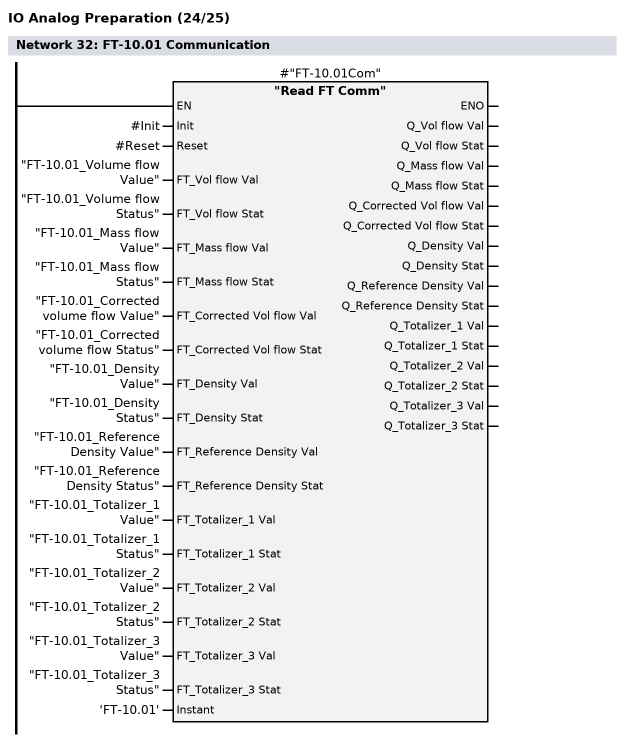
   RUNG wire#powerrail
      #"FT-10.01Com"(Init := #Init, Reset := #Reset, "FT_Vol flow Val" := "FT-10.01_Volume flow Value", "FT_Vol flow Stat" := "FT-10.01_Volume flow Status", "FT_Mass flow Val" := "FT-10.01_Mass flow Value", "FT_Mass flow Stat" := "FT-10.01_Mass flow Status", "FT_Corrected Vol flow Val" := "FT-10.01_Corrected volume flow Value", "FT_Corrected Vol flow Stat" := "FT-10.01_Corrected volume flow Status", "FT_Density Val" := "FT-10.01_Density Value", "FT_Density Stat" := "FT-10.01_Density Status", "FT_Reference Density Val" := "FT-10.01_Reference Density Value", "FT_Reference Density Stat" := "FT-10.01_Reference Density Status", "FT_Totalizer_1 Val" := "FT-10.01_Totalizer_1 Value", "FT_Totalizer_1 Stat" := "FT-10.01_Totalizer_1 Status", "FT_Totalizer_2 Val" := "FT-10.01_Totalizer_2 Value", "FT_Totalizer_2 Stat" := "FT-10.01_Totalizer_2 Status", "FT_Totalizer_3 Val" := "FT-10.01_Totalizer_3 Value", "FT_Totalizer_3 Stat" := "FT-10.01_Totalizer_3 Status", Instant := 'FT-10.01', "Q_Vol flow Val" =>, "Q_Vol flow Stat" =>, "Q_Mass flow Val" =>, "Q_Mass flow Stat" =>, "Q_Corrected Vol flow Val" =>, "Q_Corrected Vol flow Stat" =>, "Q_Density Val" =>, "Q_Density Stat" =>, "Q_Reference Density Val" =>, "Q_Reference Density Stat" =>, "Q_Totalizer_1 Val" =>, "Q_Totalizer_1 Stat" =>, "Q_Totalizer_2 Val" =>, "Q_Totalizer_2 Stat" =>, "Q_Totalizer_3 Val" =>, "Q_Totalizer_3 Stat" =>)
   END_RUNG
   // the same network as SCL:
   #"FT-10.01Com"(Init := #Init,   // "Read FT Comm"
                  Reset := #Reset,
                  "FT_Vol flow Val" := "FT-10.01_Volume flow Value",
                  "FT_Vol flow Stat" := "FT-10.01_Volume flow Status",
                  "FT_Mass flow Val" := "FT-10.01_Mass flow Value",
                  "FT_Mass flow Stat" := "FT-10.01_Mass flow Status",
                  "FT_Corrected Vol flow Val" := "FT-10.01_Corrected volume flow Value",
                  "FT_Corrected Vol flow Stat" := "FT-10.01_Corrected volume flow Status",
                  "FT_Density Val" := "FT-10.01_Density Value",
                  "FT_Density Stat" := "FT-10.01_Density Status",
                  "FT_Reference Density Val" := "FT-10.01_Reference Density Value",
                  "FT_Reference Density Stat" := "FT-10.01_Reference Density Status",
                  "FT_Totalizer_1 Val" := "FT-10.01_Totalizer_1 Value",
                  "FT_Totalizer_1 Stat" := "FT-10.01_Totalizer_1 Status",
                  "FT_Totalizer_2 Val" := "FT-10.01_Totalizer_2 Value",
                  "FT_Totalizer_2 Stat" := "FT-10.01_Totalizer_2 Status",
                  "FT_Totalizer_3 Val" := "FT-10.01_Totalizer_3 Value",
                  "FT_Totalizer_3 Stat" := "FT-10.01_Totalizer_3 Status",
                  Instant := 'FT-10.01');
END_REGION

REGION Network 33: FT-10.01 Flowrate
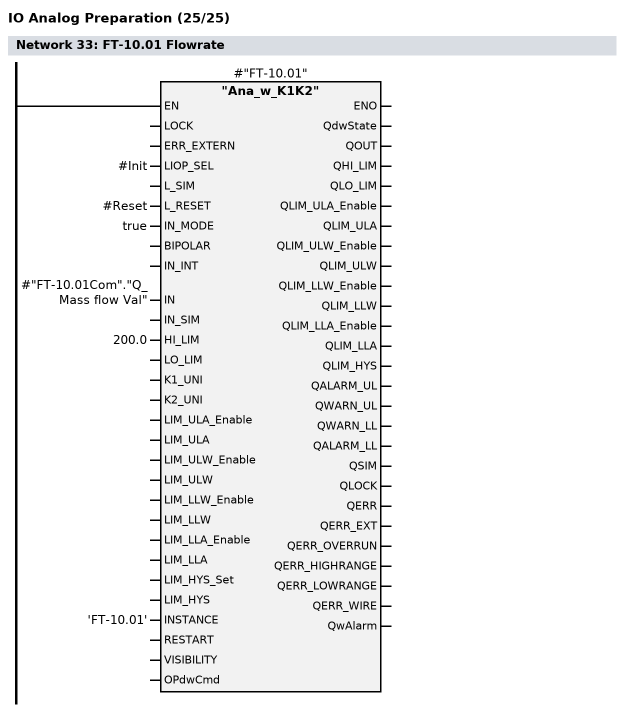
   RUNG wire#powerrail
      #"FT-10.01"(LOCK :=, ERR_EXTERN :=, LIOP_SEL := #Init, L_SIM :=, L_RESET := #Reset, IN_MODE := true, BIPOLAR :=, IN_INT :=, IN := #"FT-10.01Com"."Q_Mass flow Val", IN_SIM :=, HI_LIM := 200.0, LO_LIM :=, K1_UNI :=, K2_UNI :=, LIM_ULA_Enable :=, LIM_ULA :=, LIM_ULW_Enable :=, LIM_ULW :=, LIM_LLW_Enable :=, LIM_LLW :=, LIM_LLA_Enable :=, LIM_LLA :=, LIM_HYS_Set :=, LIM_HYS :=, INSTANCE := 'FT-10.01', RESTART :=, VISIBILITY :=, OPdwCmd :=, QdwState =>, QOUT =>, QHI_LIM =>, QLO_LIM =>, QLIM_ULA_Enable =>, QLIM_ULA =>, QLIM_ULW_Enable =>, QLIM_ULW =>, QLIM_LLW_Enable =>, QLIM_LLW =>, QLIM_LLA_Enable =>, QLIM_LLA =>, QLIM_HYS =>, QALARM_UL =>, QWARN_UL =>, QWARN_LL =>, QALARM_LL =>, QSIM =>, QLOCK =>, QERR =>, QERR_EXT =>, QERR_OVERRUN =>, QERR_HIGHRANGE =>, QERR_LOWRANGE =>, QERR_WIRE =>, QwAlarm =>)
   END_RUNG
   // the same network as SCL:
   #"FT-10.01"(LIOP_SEL := #Init,   // "Ana_w_K1K2"
               L_RESET := #Reset,
               IN_MODE := true,
               IN := #"FT-10.01Com"."Q_Mass flow Val",
               HI_LIM := 200.0,
               INSTANCE := 'FT-10.01');
END_REGION
END_FUNCTION_BLOCK

FUNCTION_BLOCK "Read FT Comm"   // FB642, LAD
{ S7_Optimized_Access := 'FALSE' }
VERSION : 0.1
// stored: AutoNumber false, IsIECCheckEnabled false, SetENOAutomatically false, UDAEnableTagReadback false
   VAR_INPUT
      Init : Bool;
      Reset : Bool;
      "FT_Vol flow Val" : Real;   // FT_Volume flow Value
      "FT_Vol flow Stat" : Byte;   // FT_Volume flow Status
      "FT_Mass flow Val" : Real;   // FT_Mass flow Value
      "FT_Mass flow Stat" : Byte;   // FT_Mass flow Status
      "FT_Corrected Vol flow Val" : Real;   // FT_Corrected volume flow Value
      "FT_Corrected Vol flow Stat" : Byte;   // FT_Corrected volume flow Status
      "FT_Density Val" : Real;   // FT_Velocity Value
      "FT_Density Stat" : Byte;   // FT_Velocity Status
      "FT_Reference Density Val" : Real;
      "FT_Reference Density Stat" : Byte;
      "FT_Totalizer_1 Val" : Real;   // FT_Totalizer_1 Value
      "FT_Totalizer_1 Stat" : Byte;   // FT_Totalizer_1 Status
      "FT_Totalizer_2 Val" : Real;   // FT_Totalizer_2 Value
      "FT_Totalizer_2 Stat" : Byte;   // FT_Totalizer_2 Status
      "FT_Totalizer_3 Val" : Real;   // FT_Totalizer_3 Value
      "FT_Totalizer_3 Stat" : Byte;   // FT_Totalizer_3 Status
      Instant { ExternalAccessible := 'False'; ExternalVisible := 'False'; ExternalWritable := 'False'} : String;
   END_VAR
   VAR_OUTPUT
      "Q_Vol flow Val" : Real;   // FT_Volume flow Value
      "Q_Vol flow Stat" : Word;   // FT_Volume flow Status
      "Q_Mass flow Val" : Real;   // FT_Mass flow Value
      "Q_Mass flow Stat" : Word;   // FT_Mass flow Status
      "Q_Corrected Vol flow Val" : Real;   // FT_Corrected volume flow Value
      "Q_Corrected Vol flow Stat" : Word;   // FT_Corrected volume flow Status
      "Q_Density Val" : Real;   // FT_Velocity Value
      "Q_Density Stat" : Word;   // FT_Velocity Status
      "Q_Reference Density Val" : Real;
      "Q_Reference Density Stat" : Word;
      "Q_Totalizer_1 Val" : Real;   // FT_Totalizer_1 Value
      "Q_Totalizer_1 Stat" : Word;   // FT_Totalizer_1 Status
      "Q_Totalizer_2 Val" : Real;   // FT_Totalizer_2 Value
      "Q_Totalizer_2 Stat" : Word;   // FT_Totalizer_2 Status
      "Q_Totalizer_3 Val" : Real;   // FT_Totalizer_3 Value
      "Q_Totalizer_3 Stat" : Word;   // FT_Totalizer_3 Status
   END_VAR
   VAR DB_SPECIFIC
      Always_On : Bool;
   END_VAR
BEGIN

REGION Network 1: Aways On
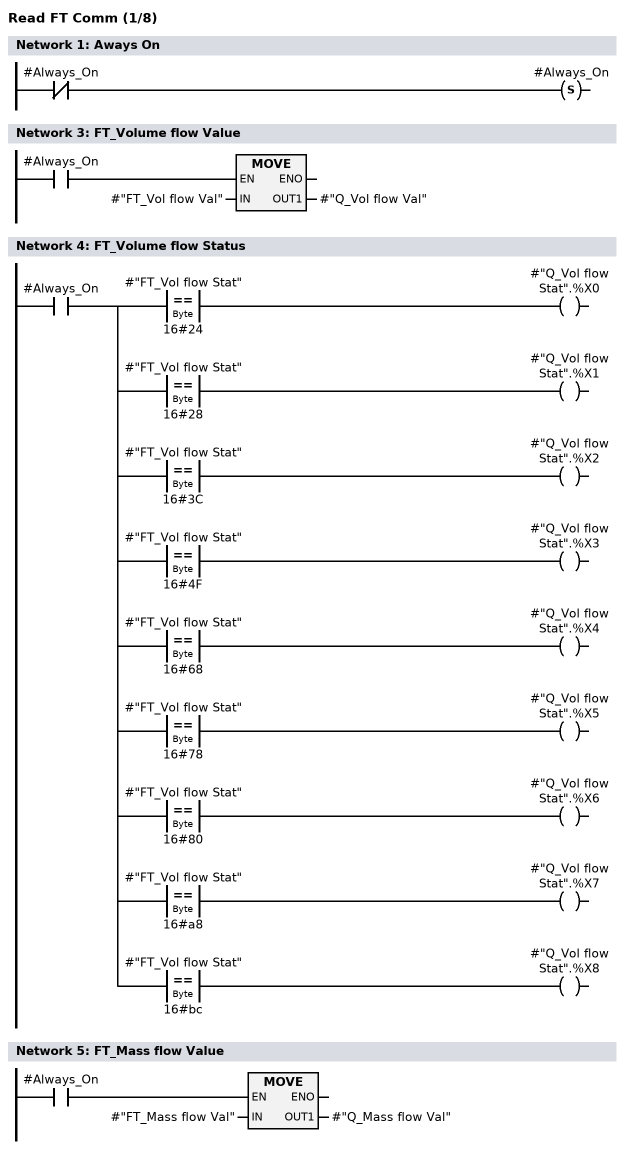
   RUNG wire#powerrail
      I_Contact( #Always_On )
      S_Coil( #Always_On )
   END_RUNG
   // the same network as SCL:
   IF NOT #Always_On THEN #Always_On := TRUE; END_IF;
END_REGION

REGION Network 2: Status Coding
   // 1. 0x24 : BAD - Maintenance alarm - A measured value is not available because a device error has occurred.
   // 2. 0x28 : BAD - Process related - A measured value is not available because the process
   // conditions are not within the device's technical specification limits.
   // 3. 0x3C : BAD - Function check - A function check is active (e.g. cleaning or calibration)
   // 4. 0x4F : UNCERTAIN - Initial value - A pre-defined value is output until a correct measured
   // value is available again or until remedial measures
   // have been carried out that change this status.
   // 5. 0x68 : UNCERTAIN - Maintenance demanded - Signs of wear and tear have been detected on the
   // measuring device. Short-term maintenance is needed to ensure that the measuring device remains
   // operational. The measured value might be invalid. The use of the measured value depends on the application.
   // 6. 0x78 : UNCERTAIN - Process related - The process conditions are not within the device's technical specification limits. This could have a negative impact on the quality and accuracy of the measured value. The use of the measured value depends on the application.
   // 7. 0x80 : GOOD - OK - No error has been diagnosed.
   // 8. 0xA8 : GOOD - Maintenance demanded -  The measured value is valid. It is highly advisable to service the device in the near future.
   // 9. 0xBC :  GOOD - Function check -  The measured value is valid. The measuring device is performing an internal function check. The function check does not have any noticeable effect on the process.
END_REGION

REGION Network 3: FT_Volume flow Value
   RUNG wire#powerrail
      Contact( #Always_On )
      Move(in := #"FT_Vol flow Val", out1 => #"Q_Vol flow Val")
   END_RUNG
   // the same network as SCL:
   IF #Always_On THEN #"Q_Vol flow Val" := #"FT_Vol flow Val"; END_IF;
END_REGION

REGION Network 4: FT_Volume flow Status
   RUNG wire#powerrail
      Contact( #Always_On )
      wire#w1
      { S7_Templates := "SrcType := Byte" } EQ_Contact(in1 := #"FT_Vol flow Stat", in2 := 16#24)
      Coil( #"Q_Vol flow Stat".%X0 )
   END_RUNG
   RUNG wire#w1
      { S7_Templates := "SrcType := Byte" } EQ_Contact(in1 := #"FT_Vol flow Stat", in2 := 16#28)
      Coil( #"Q_Vol flow Stat".%X1 )
   END_RUNG
   RUNG wire#w1
      { S7_Templates := "SrcType := Byte" } EQ_Contact(in1 := #"FT_Vol flow Stat", in2 := 16#3C)
      Coil( #"Q_Vol flow Stat".%X2 )
   END_RUNG
   RUNG wire#w1
      { S7_Templates := "SrcType := Byte" } EQ_Contact(in1 := #"FT_Vol flow Stat", in2 := 16#4F)
      Coil( #"Q_Vol flow Stat".%X3 )
   END_RUNG
   RUNG wire#w1
      { S7_Templates := "SrcType := Byte" } EQ_Contact(in1 := #"FT_Vol flow Stat", in2 := 16#68)
      Coil( #"Q_Vol flow Stat".%X4 )
   END_RUNG
   RUNG wire#w1
      { S7_Templates := "SrcType := Byte" } EQ_Contact(in1 := #"FT_Vol flow Stat", in2 := 16#78)
      Coil( #"Q_Vol flow Stat".%X5 )
   END_RUNG
   RUNG wire#w1
      { S7_Templates := "SrcType := Byte" } EQ_Contact(in1 := #"FT_Vol flow Stat", in2 := 16#80)
      Coil( #"Q_Vol flow Stat".%X6 )
   END_RUNG
   RUNG wire#w1
      { S7_Templates := "SrcType := Byte" } EQ_Contact(in1 := #"FT_Vol flow Stat", in2 := 16#a8)
      Coil( #"Q_Vol flow Stat".%X7 )
   END_RUNG
   RUNG wire#w1
      { S7_Templates := "SrcType := Byte" } EQ_Contact(in1 := #"FT_Vol flow Stat", in2 := 16#bc)
      Coil( #"Q_Vol flow Stat".%X8 )
   END_RUNG
   // the same network as SCL:
   #"Q_Vol flow Stat".%X0 := #Always_On AND (#"FT_Vol flow Stat" = 16#24);
   #"Q_Vol flow Stat".%X1 := #Always_On AND (#"FT_Vol flow Stat" = 16#28);
   #"Q_Vol flow Stat".%X2 := #Always_On AND (#"FT_Vol flow Stat" = 16#3C);
   #"Q_Vol flow Stat".%X3 := #Always_On AND (#"FT_Vol flow Stat" = 16#4F);
   #"Q_Vol flow Stat".%X4 := #Always_On AND (#"FT_Vol flow Stat" = 16#68);
   #"Q_Vol flow Stat".%X5 := #Always_On AND (#"FT_Vol flow Stat" = 16#78);
   #"Q_Vol flow Stat".%X6 := #Always_On AND (#"FT_Vol flow Stat" = 16#80);
   #"Q_Vol flow Stat".%X7 := #Always_On AND (#"FT_Vol flow Stat" = 16#a8);
   #"Q_Vol flow Stat".%X8 := #Always_On AND (#"FT_Vol flow Stat" = 16#bc);
END_REGION

REGION Network 5: FT_Mass flow Value
   RUNG wire#powerrail
      Contact( #Always_On )
      Move(in := #"FT_Mass flow Val", out1 => #"Q_Mass flow Val")
   END_RUNG
   // the same network as SCL:
   IF #Always_On THEN #"Q_Mass flow Val" := #"FT_Mass flow Val"; END_IF;
END_REGION

REGION Network 6: FT_Mass flow Status
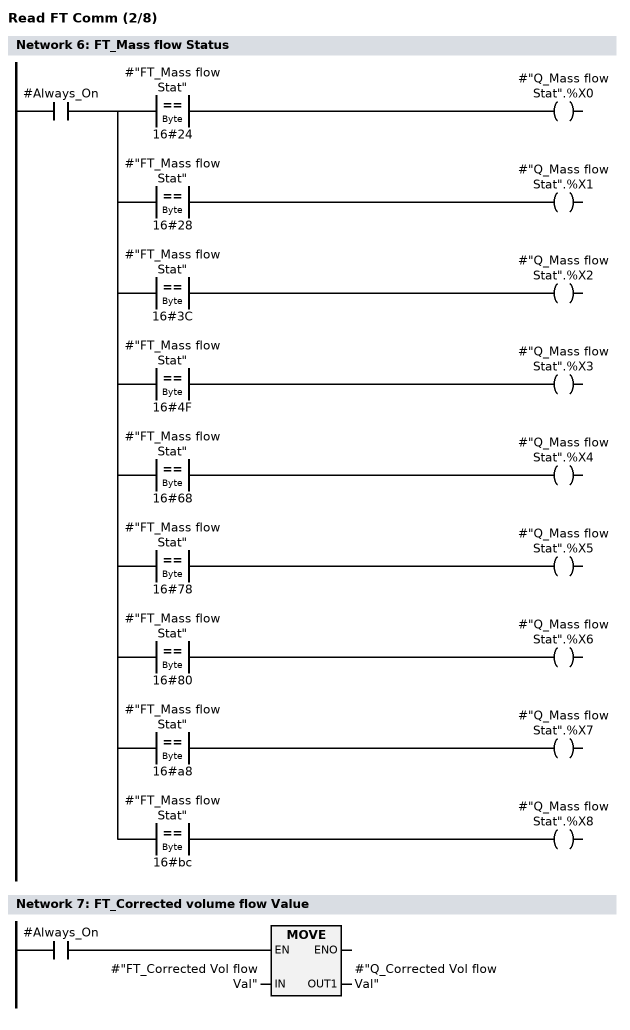
   RUNG wire#powerrail
      Contact( #Always_On )
      wire#w1
      { S7_Templates := "SrcType := Byte" } EQ_Contact(in1 := #"FT_Mass flow Stat", in2 := 16#24)
      Coil( #"Q_Mass flow Stat".%X0 )
   END_RUNG
   RUNG wire#w1
      { S7_Templates := "SrcType := Byte" } EQ_Contact(in1 := #"FT_Mass flow Stat", in2 := 16#28)
      Coil( #"Q_Mass flow Stat".%X1 )
   END_RUNG
   RUNG wire#w1
      { S7_Templates := "SrcType := Byte" } EQ_Contact(in1 := #"FT_Mass flow Stat", in2 := 16#3C)
      Coil( #"Q_Mass flow Stat".%X2 )
   END_RUNG
   RUNG wire#w1
      { S7_Templates := "SrcType := Byte" } EQ_Contact(in1 := #"FT_Mass flow Stat", in2 := 16#4F)
      Coil( #"Q_Mass flow Stat".%X3 )
   END_RUNG
   RUNG wire#w1
      { S7_Templates := "SrcType := Byte" } EQ_Contact(in1 := #"FT_Mass flow Stat", in2 := 16#68)
      Coil( #"Q_Mass flow Stat".%X4 )
   END_RUNG
   RUNG wire#w1
      { S7_Templates := "SrcType := Byte" } EQ_Contact(in1 := #"FT_Mass flow Stat", in2 := 16#78)
      Coil( #"Q_Mass flow Stat".%X5 )
   END_RUNG
   RUNG wire#w1
      { S7_Templates := "SrcType := Byte" } EQ_Contact(in1 := #"FT_Mass flow Stat", in2 := 16#80)
      Coil( #"Q_Mass flow Stat".%X6 )
   END_RUNG
   RUNG wire#w1
      { S7_Templates := "SrcType := Byte" } EQ_Contact(in1 := #"FT_Mass flow Stat", in2 := 16#a8)
      Coil( #"Q_Mass flow Stat".%X7 )
   END_RUNG
   RUNG wire#w1
      { S7_Templates := "SrcType := Byte" } EQ_Contact(in1 := #"FT_Mass flow Stat", in2 := 16#bc)
      Coil( #"Q_Mass flow Stat".%X8 )
   END_RUNG
   // the same network as SCL:
   #"Q_Mass flow Stat".%X0 := #Always_On AND (#"FT_Mass flow Stat" = 16#24);
   #"Q_Mass flow Stat".%X1 := #Always_On AND (#"FT_Mass flow Stat" = 16#28);
   #"Q_Mass flow Stat".%X2 := #Always_On AND (#"FT_Mass flow Stat" = 16#3C);
   #"Q_Mass flow Stat".%X3 := #Always_On AND (#"FT_Mass flow Stat" = 16#4F);
   #"Q_Mass flow Stat".%X4 := #Always_On AND (#"FT_Mass flow Stat" = 16#68);
   #"Q_Mass flow Stat".%X5 := #Always_On AND (#"FT_Mass flow Stat" = 16#78);
   #"Q_Mass flow Stat".%X6 := #Always_On AND (#"FT_Mass flow Stat" = 16#80);
   #"Q_Mass flow Stat".%X7 := #Always_On AND (#"FT_Mass flow Stat" = 16#a8);
   #"Q_Mass flow Stat".%X8 := #Always_On AND (#"FT_Mass flow Stat" = 16#bc);
END_REGION

REGION Network 7: FT_Corrected volume flow Value
   RUNG wire#powerrail
      Contact( #Always_On )
      Move(in := #"FT_Corrected Vol flow Val", out1 => #"Q_Corrected Vol flow Val")
   END_RUNG
   // the same network as SCL:
   IF #Always_On THEN #"Q_Corrected Vol flow Val" := #"FT_Corrected Vol flow Val"; END_IF;
END_REGION

REGION Network 8: FT_Corrected volume flow Status
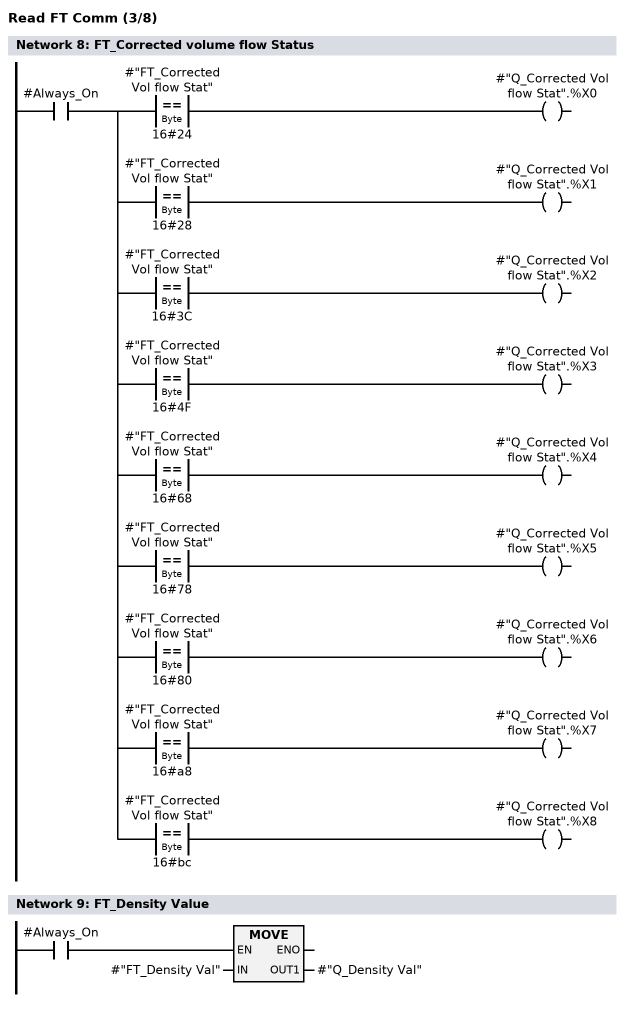
   RUNG wire#powerrail
      Contact( #Always_On )
      wire#w1
      { S7_Templates := "SrcType := Byte" } EQ_Contact(in1 := #"FT_Corrected Vol flow Stat", in2 := 16#24)
      Coil( #"Q_Corrected Vol flow Stat".%X0 )
   END_RUNG
   RUNG wire#w1
      { S7_Templates := "SrcType := Byte" } EQ_Contact(in1 := #"FT_Corrected Vol flow Stat", in2 := 16#28)
      Coil( #"Q_Corrected Vol flow Stat".%X1 )
   END_RUNG
   RUNG wire#w1
      { S7_Templates := "SrcType := Byte" } EQ_Contact(in1 := #"FT_Corrected Vol flow Stat", in2 := 16#3C)
      Coil( #"Q_Corrected Vol flow Stat".%X2 )
   END_RUNG
   RUNG wire#w1
      { S7_Templates := "SrcType := Byte" } EQ_Contact(in1 := #"FT_Corrected Vol flow Stat", in2 := 16#4F)
      Coil( #"Q_Corrected Vol flow Stat".%X3 )
   END_RUNG
   RUNG wire#w1
      { S7_Templates := "SrcType := Byte" } EQ_Contact(in1 := #"FT_Corrected Vol flow Stat", in2 := 16#68)
      Coil( #"Q_Corrected Vol flow Stat".%X4 )
   END_RUNG
   RUNG wire#w1
      { S7_Templates := "SrcType := Byte" } EQ_Contact(in1 := #"FT_Corrected Vol flow Stat", in2 := 16#78)
      Coil( #"Q_Corrected Vol flow Stat".%X5 )
   END_RUNG
   RUNG wire#w1
      { S7_Templates := "SrcType := Byte" } EQ_Contact(in1 := #"FT_Corrected Vol flow Stat", in2 := 16#80)
      Coil( #"Q_Corrected Vol flow Stat".%X6 )
   END_RUNG
   RUNG wire#w1
      { S7_Templates := "SrcType := Byte" } EQ_Contact(in1 := #"FT_Corrected Vol flow Stat", in2 := 16#a8)
      Coil( #"Q_Corrected Vol flow Stat".%X7 )
   END_RUNG
   RUNG wire#w1
      { S7_Templates := "SrcType := Byte" } EQ_Contact(in1 := #"FT_Corrected Vol flow Stat", in2 := 16#bc)
      Coil( #"Q_Corrected Vol flow Stat".%X8 )
   END_RUNG
   // the same network as SCL:
   #"Q_Corrected Vol flow Stat".%X0 := #Always_On AND (#"FT_Corrected Vol flow Stat" = 16#24);
   #"Q_Corrected Vol flow Stat".%X1 := #Always_On AND (#"FT_Corrected Vol flow Stat" = 16#28);
   #"Q_Corrected Vol flow Stat".%X2 := #Always_On AND (#"FT_Corrected Vol flow Stat" = 16#3C);
   #"Q_Corrected Vol flow Stat".%X3 := #Always_On AND (#"FT_Corrected Vol flow Stat" = 16#4F);
   #"Q_Corrected Vol flow Stat".%X4 := #Always_On AND (#"FT_Corrected Vol flow Stat" = 16#68);
   #"Q_Corrected Vol flow Stat".%X5 := #Always_On AND (#"FT_Corrected Vol flow Stat" = 16#78);
   #"Q_Corrected Vol flow Stat".%X6 := #Always_On AND (#"FT_Corrected Vol flow Stat" = 16#80);
   #"Q_Corrected Vol flow Stat".%X7 := #Always_On AND (#"FT_Corrected Vol flow Stat" = 16#a8);
   #"Q_Corrected Vol flow Stat".%X8 := #Always_On AND (#"FT_Corrected Vol flow Stat" = 16#bc);
END_REGION

REGION Network 9: FT_Density Value
   RUNG wire#powerrail
      Contact( #Always_On )
      Move(in := #"FT_Density Val", out1 => #"Q_Density Val")
   END_RUNG
   // the same network as SCL:
   IF #Always_On THEN #"Q_Density Val" := #"FT_Density Val"; END_IF;
END_REGION

REGION Network 10: FT_Density Status
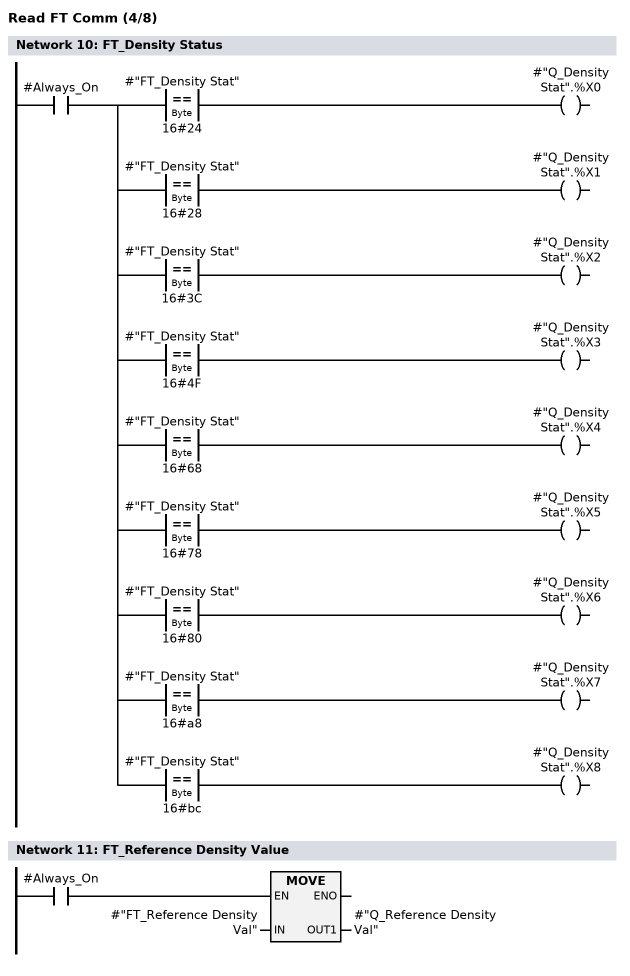
   RUNG wire#powerrail
      Contact( #Always_On )
      wire#w1
      { S7_Templates := "SrcType := Byte" } EQ_Contact(in1 := #"FT_Density Stat", in2 := 16#24)
      Coil( #"Q_Density Stat".%X0 )
   END_RUNG
   RUNG wire#w1
      { S7_Templates := "SrcType := Byte" } EQ_Contact(in1 := #"FT_Density Stat", in2 := 16#28)
      Coil( #"Q_Density Stat".%X1 )
   END_RUNG
   RUNG wire#w1
      { S7_Templates := "SrcType := Byte" } EQ_Contact(in1 := #"FT_Density Stat", in2 := 16#3C)
      Coil( #"Q_Density Stat".%X2 )
   END_RUNG
   RUNG wire#w1
      { S7_Templates := "SrcType := Byte" } EQ_Contact(in1 := #"FT_Density Stat", in2 := 16#4F)
      Coil( #"Q_Density Stat".%X3 )
   END_RUNG
   RUNG wire#w1
      { S7_Templates := "SrcType := Byte" } EQ_Contact(in1 := #"FT_Density Stat", in2 := 16#68)
      Coil( #"Q_Density Stat".%X4 )
   END_RUNG
   RUNG wire#w1
      { S7_Templates := "SrcType := Byte" } EQ_Contact(in1 := #"FT_Density Stat", in2 := 16#78)
      Coil( #"Q_Density Stat".%X5 )
   END_RUNG
   RUNG wire#w1
      { S7_Templates := "SrcType := Byte" } EQ_Contact(in1 := #"FT_Density Stat", in2 := 16#80)
      Coil( #"Q_Density Stat".%X6 )
   END_RUNG
   RUNG wire#w1
      { S7_Templates := "SrcType := Byte" } EQ_Contact(in1 := #"FT_Density Stat", in2 := 16#a8)
      Coil( #"Q_Density Stat".%X7 )
   END_RUNG
   RUNG wire#w1
      { S7_Templates := "SrcType := Byte" } EQ_Contact(in1 := #"FT_Density Stat", in2 := 16#bc)
      Coil( #"Q_Density Stat".%X8 )
   END_RUNG
   // the same network as SCL:
   #"Q_Density Stat".%X0 := #Always_On AND (#"FT_Density Stat" = 16#24);
   #"Q_Density Stat".%X1 := #Always_On AND (#"FT_Density Stat" = 16#28);
   #"Q_Density Stat".%X2 := #Always_On AND (#"FT_Density Stat" = 16#3C);
   #"Q_Density Stat".%X3 := #Always_On AND (#"FT_Density Stat" = 16#4F);
   #"Q_Density Stat".%X4 := #Always_On AND (#"FT_Density Stat" = 16#68);
   #"Q_Density Stat".%X5 := #Always_On AND (#"FT_Density Stat" = 16#78);
   #"Q_Density Stat".%X6 := #Always_On AND (#"FT_Density Stat" = 16#80);
   #"Q_Density Stat".%X7 := #Always_On AND (#"FT_Density Stat" = 16#a8);
   #"Q_Density Stat".%X8 := #Always_On AND (#"FT_Density Stat" = 16#bc);
END_REGION

REGION Network 11: FT_Reference Density Value
   RUNG wire#powerrail
      Contact( #Always_On )
      Move(in := #"FT_Reference Density Val", out1 => #"Q_Reference Density Val")
   END_RUNG
   // the same network as SCL:
   IF #Always_On THEN #"Q_Reference Density Val" := #"FT_Reference Density Val"; END_IF;
END_REGION

REGION Network 12: FT_Reference Density Status
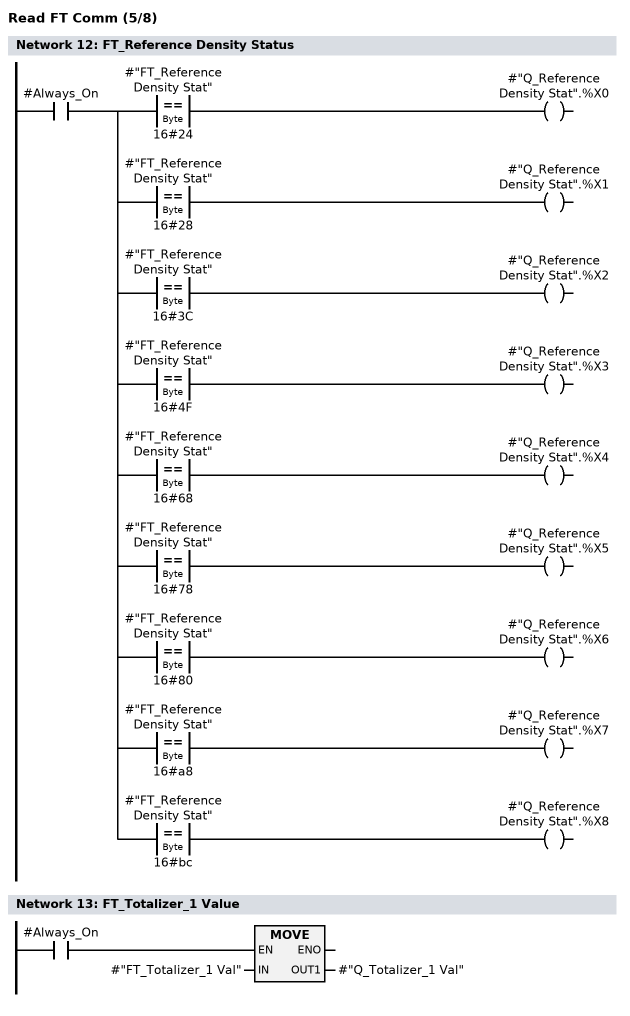
   RUNG wire#powerrail
      Contact( #Always_On )
      wire#w1
      { S7_Templates := "SrcType := Byte" } EQ_Contact(in1 := #"FT_Reference Density Stat", in2 := 16#24)
      Coil( #"Q_Reference Density Stat".%X0 )
   END_RUNG
   RUNG wire#w1
      { S7_Templates := "SrcType := Byte" } EQ_Contact(in1 := #"FT_Reference Density Stat", in2 := 16#28)
      Coil( #"Q_Reference Density Stat".%X1 )
   END_RUNG
   RUNG wire#w1
      { S7_Templates := "SrcType := Byte" } EQ_Contact(in1 := #"FT_Reference Density Stat", in2 := 16#3C)
      Coil( #"Q_Reference Density Stat".%X2 )
   END_RUNG
   RUNG wire#w1
      { S7_Templates := "SrcType := Byte" } EQ_Contact(in1 := #"FT_Reference Density Stat", in2 := 16#4F)
      Coil( #"Q_Reference Density Stat".%X3 )
   END_RUNG
   RUNG wire#w1
      { S7_Templates := "SrcType := Byte" } EQ_Contact(in1 := #"FT_Reference Density Stat", in2 := 16#68)
      Coil( #"Q_Reference Density Stat".%X4 )
   END_RUNG
   RUNG wire#w1
      { S7_Templates := "SrcType := Byte" } EQ_Contact(in1 := #"FT_Reference Density Stat", in2 := 16#78)
      Coil( #"Q_Reference Density Stat".%X5 )
   END_RUNG
   RUNG wire#w1
      { S7_Templates := "SrcType := Byte" } EQ_Contact(in1 := #"FT_Reference Density Stat", in2 := 16#80)
      Coil( #"Q_Reference Density Stat".%X6 )
   END_RUNG
   RUNG wire#w1
      { S7_Templates := "SrcType := Byte" } EQ_Contact(in1 := #"FT_Reference Density Stat", in2 := 16#a8)
      Coil( #"Q_Reference Density Stat".%X7 )
   END_RUNG
   RUNG wire#w1
      { S7_Templates := "SrcType := Byte" } EQ_Contact(in1 := #"FT_Reference Density Stat", in2 := 16#bc)
      Coil( #"Q_Reference Density Stat".%X8 )
   END_RUNG
   // the same network as SCL:
   #"Q_Reference Density Stat".%X0 := #Always_On AND (#"FT_Reference Density Stat" = 16#24);
   #"Q_Reference Density Stat".%X1 := #Always_On AND (#"FT_Reference Density Stat" = 16#28);
   #"Q_Reference Density Stat".%X2 := #Always_On AND (#"FT_Reference Density Stat" = 16#3C);
   #"Q_Reference Density Stat".%X3 := #Always_On AND (#"FT_Reference Density Stat" = 16#4F);
   #"Q_Reference Density Stat".%X4 := #Always_On AND (#"FT_Reference Density Stat" = 16#68);
   #"Q_Reference Density Stat".%X5 := #Always_On AND (#"FT_Reference Density Stat" = 16#78);
   #"Q_Reference Density Stat".%X6 := #Always_On AND (#"FT_Reference Density Stat" = 16#80);
   #"Q_Reference Density Stat".%X7 := #Always_On AND (#"FT_Reference Density Stat" = 16#a8);
   #"Q_Reference Density Stat".%X8 := #Always_On AND (#"FT_Reference Density Stat" = 16#bc);
END_REGION

REGION Network 13: FT_Totalizer_1 Value
   RUNG wire#powerrail
      Contact( #Always_On )
      Move(in := #"FT_Totalizer_1 Val", out1 => #"Q_Totalizer_1 Val")
   END_RUNG
   // the same network as SCL:
   IF #Always_On THEN #"Q_Totalizer_1 Val" := #"FT_Totalizer_1 Val"; END_IF;
END_REGION

REGION Network 14: FT_Totalizer_1 Status
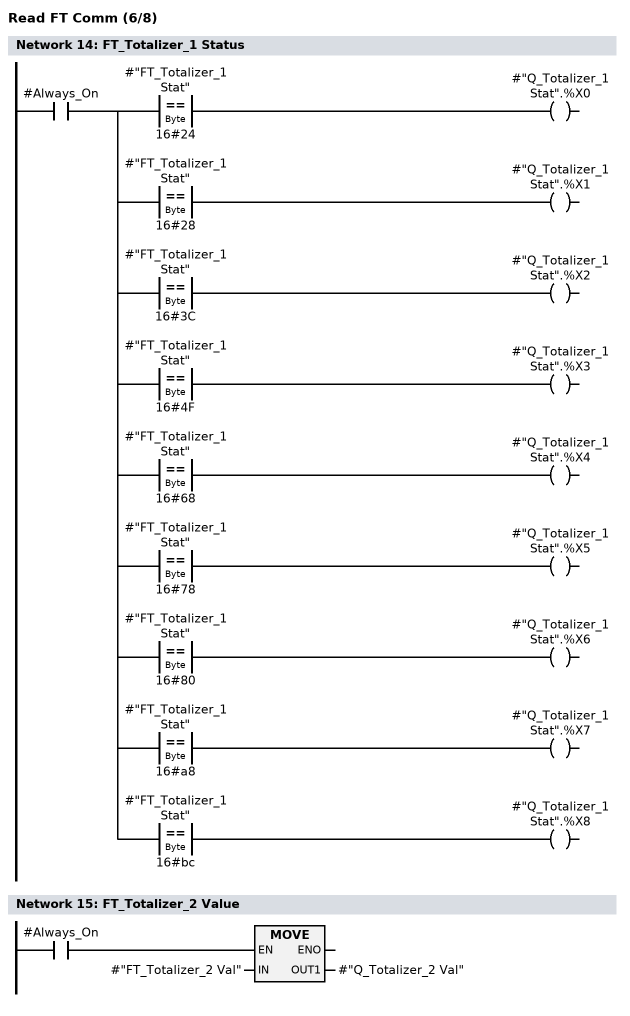
   RUNG wire#powerrail
      Contact( #Always_On )
      wire#w1
      { S7_Templates := "SrcType := Byte" } EQ_Contact(in1 := #"FT_Totalizer_1 Stat", in2 := 16#24)
      Coil( #"Q_Totalizer_1 Stat".%X0 )
   END_RUNG
   RUNG wire#w1
      { S7_Templates := "SrcType := Byte" } EQ_Contact(in1 := #"FT_Totalizer_1 Stat", in2 := 16#28)
      Coil( #"Q_Totalizer_1 Stat".%X1 )
   END_RUNG
   RUNG wire#w1
      { S7_Templates := "SrcType := Byte" } EQ_Contact(in1 := #"FT_Totalizer_1 Stat", in2 := 16#3C)
      Coil( #"Q_Totalizer_1 Stat".%X2 )
   END_RUNG
   RUNG wire#w1
      { S7_Templates := "SrcType := Byte" } EQ_Contact(in1 := #"FT_Totalizer_1 Stat", in2 := 16#4F)
      Coil( #"Q_Totalizer_1 Stat".%X3 )
   END_RUNG
   RUNG wire#w1
      { S7_Templates := "SrcType := Byte" } EQ_Contact(in1 := #"FT_Totalizer_1 Stat", in2 := 16#68)
      Coil( #"Q_Totalizer_1 Stat".%X4 )
   END_RUNG
   RUNG wire#w1
      { S7_Templates := "SrcType := Byte" } EQ_Contact(in1 := #"FT_Totalizer_1 Stat", in2 := 16#78)
      Coil( #"Q_Totalizer_1 Stat".%X5 )
   END_RUNG
   RUNG wire#w1
      { S7_Templates := "SrcType := Byte" } EQ_Contact(in1 := #"FT_Totalizer_1 Stat", in2 := 16#80)
      Coil( #"Q_Totalizer_1 Stat".%X6 )
   END_RUNG
   RUNG wire#w1
      { S7_Templates := "SrcType := Byte" } EQ_Contact(in1 := #"FT_Totalizer_1 Stat", in2 := 16#a8)
      Coil( #"Q_Totalizer_1 Stat".%X7 )
   END_RUNG
   RUNG wire#w1
      { S7_Templates := "SrcType := Byte" } EQ_Contact(in1 := #"FT_Totalizer_1 Stat", in2 := 16#bc)
      Coil( #"Q_Totalizer_1 Stat".%X8 )
   END_RUNG
   // the same network as SCL:
   #"Q_Totalizer_1 Stat".%X0 := #Always_On AND (#"FT_Totalizer_1 Stat" = 16#24);
   #"Q_Totalizer_1 Stat".%X1 := #Always_On AND (#"FT_Totalizer_1 Stat" = 16#28);
   #"Q_Totalizer_1 Stat".%X2 := #Always_On AND (#"FT_Totalizer_1 Stat" = 16#3C);
   #"Q_Totalizer_1 Stat".%X3 := #Always_On AND (#"FT_Totalizer_1 Stat" = 16#4F);
   #"Q_Totalizer_1 Stat".%X4 := #Always_On AND (#"FT_Totalizer_1 Stat" = 16#68);
   #"Q_Totalizer_1 Stat".%X5 := #Always_On AND (#"FT_Totalizer_1 Stat" = 16#78);
   #"Q_Totalizer_1 Stat".%X6 := #Always_On AND (#"FT_Totalizer_1 Stat" = 16#80);
   #"Q_Totalizer_1 Stat".%X7 := #Always_On AND (#"FT_Totalizer_1 Stat" = 16#a8);
   #"Q_Totalizer_1 Stat".%X8 := #Always_On AND (#"FT_Totalizer_1 Stat" = 16#bc);
END_REGION

REGION Network 15: FT_Totalizer_2 Value
   RUNG wire#powerrail
      Contact( #Always_On )
      Move(in := #"FT_Totalizer_2 Val", out1 => #"Q_Totalizer_2 Val")
   END_RUNG
   // the same network as SCL:
   IF #Always_On THEN #"Q_Totalizer_2 Val" := #"FT_Totalizer_2 Val"; END_IF;
END_REGION

REGION Network 16: FT_Totalizer_2 Status
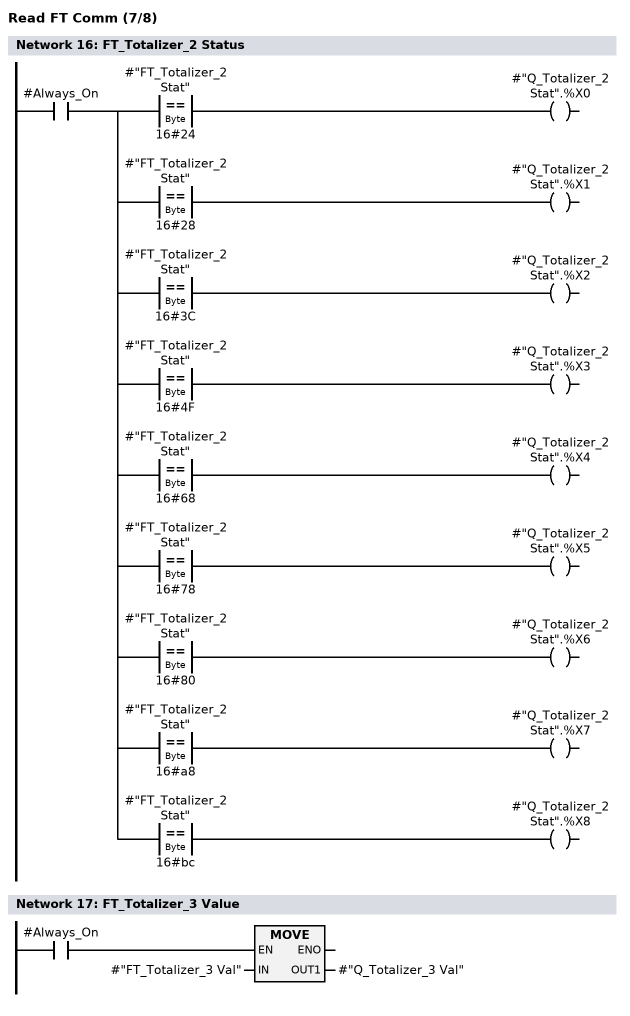
   RUNG wire#powerrail
      Contact( #Always_On )
      wire#w1
      { S7_Templates := "SrcType := Byte" } EQ_Contact(in1 := #"FT_Totalizer_2 Stat", in2 := 16#24)
      Coil( #"Q_Totalizer_2 Stat".%X0 )
   END_RUNG
   RUNG wire#w1
      { S7_Templates := "SrcType := Byte" } EQ_Contact(in1 := #"FT_Totalizer_2 Stat", in2 := 16#28)
      Coil( #"Q_Totalizer_2 Stat".%X1 )
   END_RUNG
   RUNG wire#w1
      { S7_Templates := "SrcType := Byte" } EQ_Contact(in1 := #"FT_Totalizer_2 Stat", in2 := 16#3C)
      Coil( #"Q_Totalizer_2 Stat".%X2 )
   END_RUNG
   RUNG wire#w1
      { S7_Templates := "SrcType := Byte" } EQ_Contact(in1 := #"FT_Totalizer_2 Stat", in2 := 16#4F)
      Coil( #"Q_Totalizer_2 Stat".%X3 )
   END_RUNG
   RUNG wire#w1
      { S7_Templates := "SrcType := Byte" } EQ_Contact(in1 := #"FT_Totalizer_2 Stat", in2 := 16#68)
      Coil( #"Q_Totalizer_2 Stat".%X4 )
   END_RUNG
   RUNG wire#w1
      { S7_Templates := "SrcType := Byte" } EQ_Contact(in1 := #"FT_Totalizer_2 Stat", in2 := 16#78)
      Coil( #"Q_Totalizer_2 Stat".%X5 )
   END_RUNG
   RUNG wire#w1
      { S7_Templates := "SrcType := Byte" } EQ_Contact(in1 := #"FT_Totalizer_2 Stat", in2 := 16#80)
      Coil( #"Q_Totalizer_2 Stat".%X6 )
   END_RUNG
   RUNG wire#w1
      { S7_Templates := "SrcType := Byte" } EQ_Contact(in1 := #"FT_Totalizer_2 Stat", in2 := 16#a8)
      Coil( #"Q_Totalizer_2 Stat".%X7 )
   END_RUNG
   RUNG wire#w1
      { S7_Templates := "SrcType := Byte" } EQ_Contact(in1 := #"FT_Totalizer_2 Stat", in2 := 16#bc)
      Coil( #"Q_Totalizer_2 Stat".%X8 )
   END_RUNG
   // the same network as SCL:
   #"Q_Totalizer_2 Stat".%X0 := #Always_On AND (#"FT_Totalizer_2 Stat" = 16#24);
   #"Q_Totalizer_2 Stat".%X1 := #Always_On AND (#"FT_Totalizer_2 Stat" = 16#28);
   #"Q_Totalizer_2 Stat".%X2 := #Always_On AND (#"FT_Totalizer_2 Stat" = 16#3C);
   #"Q_Totalizer_2 Stat".%X3 := #Always_On AND (#"FT_Totalizer_2 Stat" = 16#4F);
   #"Q_Totalizer_2 Stat".%X4 := #Always_On AND (#"FT_Totalizer_2 Stat" = 16#68);
   #"Q_Totalizer_2 Stat".%X5 := #Always_On AND (#"FT_Totalizer_2 Stat" = 16#78);
   #"Q_Totalizer_2 Stat".%X6 := #Always_On AND (#"FT_Totalizer_2 Stat" = 16#80);
   #"Q_Totalizer_2 Stat".%X7 := #Always_On AND (#"FT_Totalizer_2 Stat" = 16#a8);
   #"Q_Totalizer_2 Stat".%X8 := #Always_On AND (#"FT_Totalizer_2 Stat" = 16#bc);
END_REGION

REGION Network 17: FT_Totalizer_3 Value
   RUNG wire#powerrail
      Contact( #Always_On )
      Move(in := #"FT_Totalizer_3 Val", out1 => #"Q_Totalizer_3 Val")
   END_RUNG
   // the same network as SCL:
   IF #Always_On THEN #"Q_Totalizer_3 Val" := #"FT_Totalizer_3 Val"; END_IF;
END_REGION

REGION Network 18: FT_Totalizer_3 Status
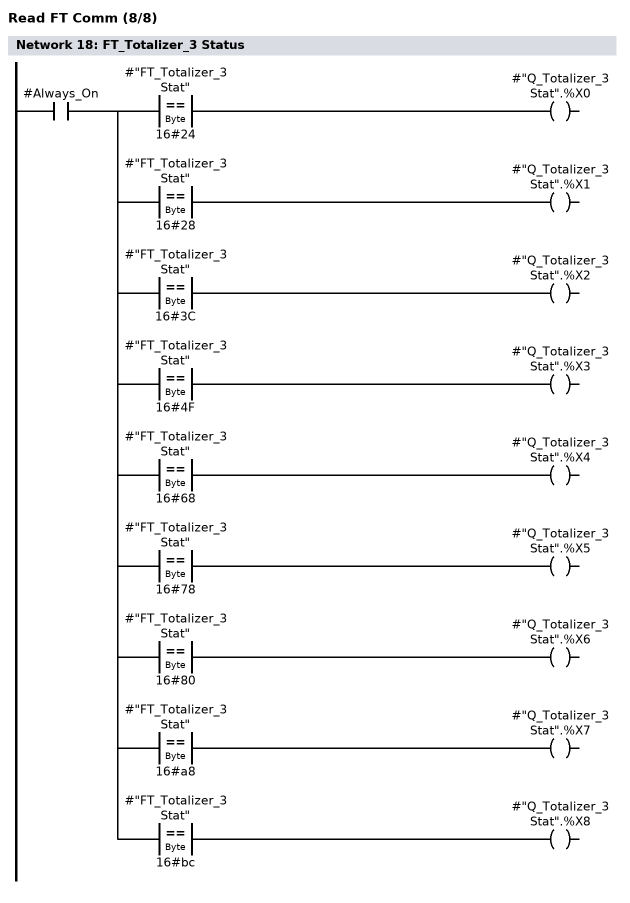
   RUNG wire#powerrail
      Contact( #Always_On )
      wire#w1
      { S7_Templates := "SrcType := Byte" } EQ_Contact(in1 := #"FT_Totalizer_3 Stat", in2 := 16#24)
      Coil( #"Q_Totalizer_3 Stat".%X0 )
   END_RUNG
   RUNG wire#w1
      { S7_Templates := "SrcType := Byte" } EQ_Contact(in1 := #"FT_Totalizer_3 Stat", in2 := 16#28)
      Coil( #"Q_Totalizer_3 Stat".%X1 )
   END_RUNG
   RUNG wire#w1
      { S7_Templates := "SrcType := Byte" } EQ_Contact(in1 := #"FT_Totalizer_3 Stat", in2 := 16#3C)
      Coil( #"Q_Totalizer_3 Stat".%X2 )
   END_RUNG
   RUNG wire#w1
      { S7_Templates := "SrcType := Byte" } EQ_Contact(in1 := #"FT_Totalizer_3 Stat", in2 := 16#4F)
      Coil( #"Q_Totalizer_3 Stat".%X3 )
   END_RUNG
   RUNG wire#w1
      { S7_Templates := "SrcType := Byte" } EQ_Contact(in1 := #"FT_Totalizer_3 Stat", in2 := 16#68)
      Coil( #"Q_Totalizer_3 Stat".%X4 )
   END_RUNG
   RUNG wire#w1
      { S7_Templates := "SrcType := Byte" } EQ_Contact(in1 := #"FT_Totalizer_3 Stat", in2 := 16#78)
      Coil( #"Q_Totalizer_3 Stat".%X5 )
   END_RUNG
   RUNG wire#w1
      { S7_Templates := "SrcType := Byte" } EQ_Contact(in1 := #"FT_Totalizer_3 Stat", in2 := 16#80)
      Coil( #"Q_Totalizer_3 Stat".%X6 )
   END_RUNG
   RUNG wire#w1
      { S7_Templates := "SrcType := Byte" } EQ_Contact(in1 := #"FT_Totalizer_3 Stat", in2 := 16#a8)
      Coil( #"Q_Totalizer_3 Stat".%X7 )
   END_RUNG
   RUNG wire#w1
      { S7_Templates := "SrcType := Byte" } EQ_Contact(in1 := #"FT_Totalizer_3 Stat", in2 := 16#bc)
      Coil( #"Q_Totalizer_3 Stat".%X8 )
   END_RUNG
   // the same network as SCL:
   #"Q_Totalizer_3 Stat".%X0 := #Always_On AND (#"FT_Totalizer_3 Stat" = 16#24);
   #"Q_Totalizer_3 Stat".%X1 := #Always_On AND (#"FT_Totalizer_3 Stat" = 16#28);
   #"Q_Totalizer_3 Stat".%X2 := #Always_On AND (#"FT_Totalizer_3 Stat" = 16#3C);
   #"Q_Totalizer_3 Stat".%X3 := #Always_On AND (#"FT_Totalizer_3 Stat" = 16#4F);
   #"Q_Totalizer_3 Stat".%X4 := #Always_On AND (#"FT_Totalizer_3 Stat" = 16#68);
   #"Q_Totalizer_3 Stat".%X5 := #Always_On AND (#"FT_Totalizer_3 Stat" = 16#78);
   #"Q_Totalizer_3 Stat".%X6 := #Always_On AND (#"FT_Totalizer_3 Stat" = 16#80);
   #"Q_Totalizer_3 Stat".%X7 := #Always_On AND (#"FT_Totalizer_3 Stat" = 16#a8);
   #"Q_Totalizer_3 Stat".%X8 := #Always_On AND (#"FT_Totalizer_3 Stat" = 16#bc);
END_REGION
END_FUNCTION_BLOCK

FUNCTION_BLOCK "IO Digital Preparation"   // FB8, LAD
{ S7_Optimized_Access := 'FALSE' }
VERSION : 0.1
// stored: AutoNumber true, IsIECCheckEnabled false, SetENOAutomatically false, UDAEnableTagReadback false
   VAR_INPUT
      init : Bool;
      Reset : Bool;
   END_VAR
   VAR
      "FS-01.01" { S7_SetPoint := 'True'} : "Digital";   // FLOW SWITCH LINE HOT WATER PHE-01.01
      "DRP-P02.01" { S7_SetPoint := 'True'} : "Digital";   // DRY RUN PROTECTION MONO PUMP P-02.01
      "DRP-P02.02" { S7_SetPoint := 'True'} : "Digital";   // DRY RUN PROTECTION MONO PUMP P-02.03
      "DRP-P03.01" { S7_SetPoint := 'True'} : "Digital";   // DRY RUN PROTECTION MONO PUMP P-03.01
      "DRP-P03.02" { S7_SetPoint := 'True'} : "Digital";   // DRY RUN PROTECTION MONO PUMP P-03.03
      "DRP-P04.01" { S7_SetPoint := 'True'} : "Digital";   // DRY RUN PROTECTION MONO PUMP P-04.01
      "DRP-P05.01" { S7_SetPoint := 'True'} : "Digital";   // DRY RUN PROTECTION MONO PUMP P-05.01
      "DRP-P05.02" { S7_SetPoint := 'True'} : "Digital";   // DRY RUN PROTECTION MONO PUMP P-05.03
      "DRP-P06.01" { S7_SetPoint := 'True'} : "Digital";   // DRY RUN PROTECTION MONO PUMP P-06.01
      "DRP-P07.01" { S7_SetPoint := 'True'} : "Digital";   // DRY RUN PROTECTION MONO PUMP P-07.01
      "DRP-P08.01" { S7_SetPoint := 'True'} : "Digital";   // DRY RUN PROTECTION MONO PUMP P-08.01
      "DRP-P09.01" { S7_SetPoint := 'True'} : "Digital";   // DRY RUN PROTECTION MONO PUMP P-09.01
      "DRP-P09.02" { S7_SetPoint := 'True'} : "Digital";   // DRY RUN PROTECTION MONO PUMP P-09.03
      "LL-51.01" { S7_SetPoint := 'True'} : "Digital";
      "ML-51.01" { S7_SetPoint := 'True'} : "Digital";
      "HL-51.01" { S7_SetPoint := 'True'} : "Digital";
   END_VAR
BEGIN

REGION Network 1: FS-01.01
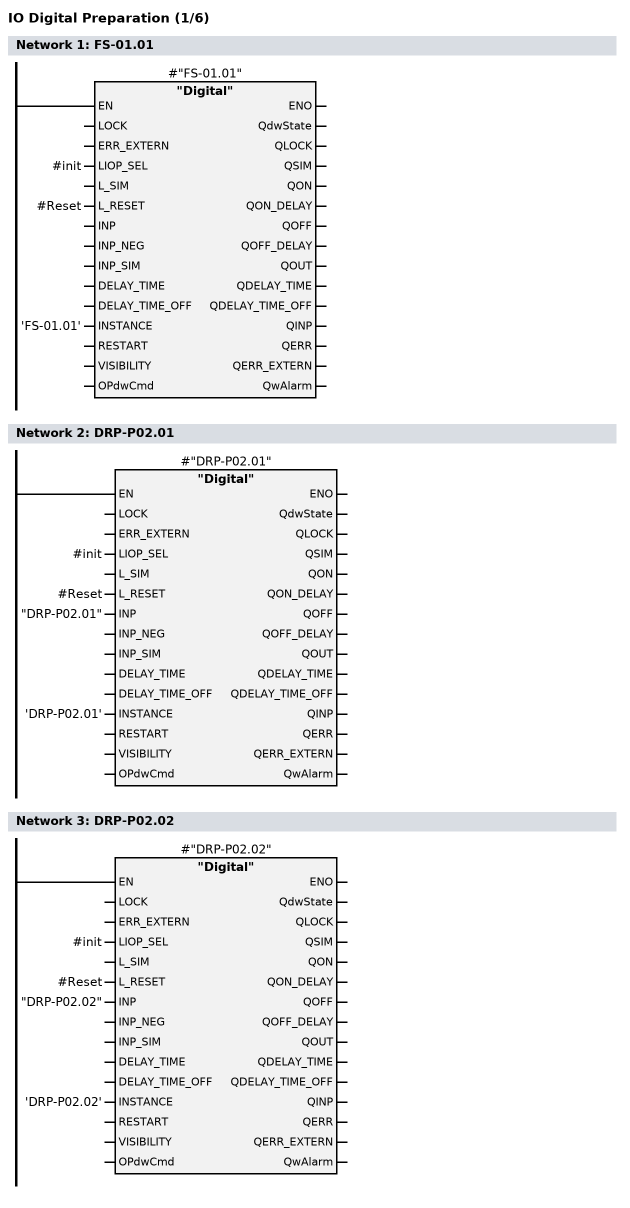
   RUNG wire#powerrail
      #"FS-01.01"(LOCK :=, ERR_EXTERN :=, LIOP_SEL := #init, L_SIM :=, L_RESET := #Reset, INP :=, INP_NEG :=, INP_SIM :=, DELAY_TIME :=, DELAY_TIME_OFF :=, INSTANCE := 'FS-01.01', RESTART :=, VISIBILITY :=, OPdwCmd :=, QdwState =>, QLOCK =>, QSIM =>, QON =>, QON_DELAY =>, QOFF =>, QOFF_DELAY =>, QOUT =>, QDELAY_TIME =>, QDELAY_TIME_OFF =>, QINP =>, QERR =>, QERR_EXTERN =>, QwAlarm =>)
   END_RUNG
   // the same network as SCL:
   #"FS-01.01"(LIOP_SEL := #init, L_RESET := #Reset, INSTANCE := 'FS-01.01');   // "Digital"
END_REGION

REGION Network 2: DRP-P02.01
   RUNG wire#powerrail
      #"DRP-P02.01"(LOCK :=, ERR_EXTERN :=, LIOP_SEL := #init, L_SIM :=, L_RESET := #Reset, INP := "DRP-P02.01", INP_NEG :=, INP_SIM :=, DELAY_TIME :=, DELAY_TIME_OFF :=, INSTANCE := 'DRP-P02.01', RESTART :=, VISIBILITY :=, OPdwCmd :=, QdwState =>, QLOCK =>, QSIM =>, QON =>, QON_DELAY =>, QOFF =>, QOFF_DELAY =>, QOUT =>, QDELAY_TIME =>, QDELAY_TIME_OFF =>, QINP =>, QERR =>, QERR_EXTERN =>, QwAlarm =>)
   END_RUNG
   // the same network as SCL:
   #"DRP-P02.01"(LIOP_SEL := #init, L_RESET := #Reset, INP := "DRP-P02.01", INSTANCE := 'DRP-P02.01');   // "Digital"
END_REGION

REGION Network 3: DRP-P02.02
   RUNG wire#powerrail
      #"DRP-P02.02"(LOCK :=, ERR_EXTERN :=, LIOP_SEL := #init, L_SIM :=, L_RESET := #Reset, INP := "DRP-P02.02", INP_NEG :=, INP_SIM :=, DELAY_TIME :=, DELAY_TIME_OFF :=, INSTANCE := 'DRP-P02.02', RESTART :=, VISIBILITY :=, OPdwCmd :=, QdwState =>, QLOCK =>, QSIM =>, QON =>, QON_DELAY =>, QOFF =>, QOFF_DELAY =>, QOUT =>, QDELAY_TIME =>, QDELAY_TIME_OFF =>, QINP =>, QERR =>, QERR_EXTERN =>, QwAlarm =>)
   END_RUNG
   // the same network as SCL:
   #"DRP-P02.02"(LIOP_SEL := #init, L_RESET := #Reset, INP := "DRP-P02.02", INSTANCE := 'DRP-P02.02');   // "Digital"
END_REGION

REGION Network 4: DRP-P03.01
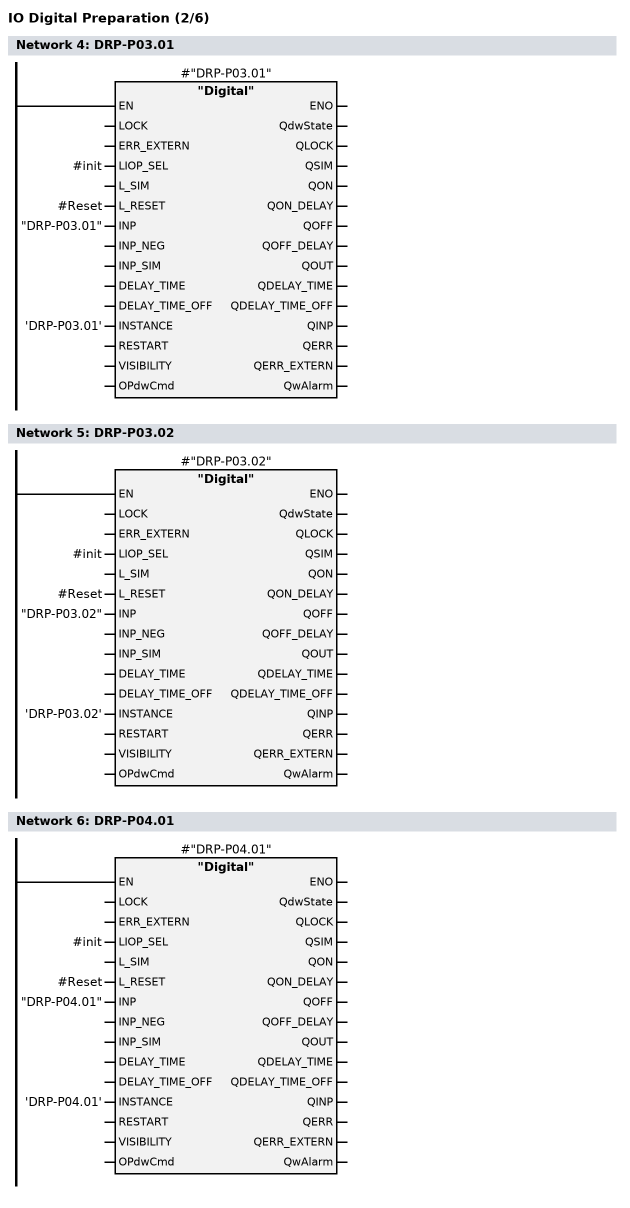
   RUNG wire#powerrail
      #"DRP-P03.01"(LOCK :=, ERR_EXTERN :=, LIOP_SEL := #init, L_SIM :=, L_RESET := #Reset, INP := "DRP-P03.01", INP_NEG :=, INP_SIM :=, DELAY_TIME :=, DELAY_TIME_OFF :=, INSTANCE := 'DRP-P03.01', RESTART :=, VISIBILITY :=, OPdwCmd :=, QdwState =>, QLOCK =>, QSIM =>, QON =>, QON_DELAY =>, QOFF =>, QOFF_DELAY =>, QOUT =>, QDELAY_TIME =>, QDELAY_TIME_OFF =>, QINP =>, QERR =>, QERR_EXTERN =>, QwAlarm =>)
   END_RUNG
   // the same network as SCL:
   #"DRP-P03.01"(LIOP_SEL := #init, L_RESET := #Reset, INP := "DRP-P03.01", INSTANCE := 'DRP-P03.01');   // "Digital"
END_REGION

REGION Network 5: DRP-P03.02
   RUNG wire#powerrail
      #"DRP-P03.02"(LOCK :=, ERR_EXTERN :=, LIOP_SEL := #init, L_SIM :=, L_RESET := #Reset, INP := "DRP-P03.02", INP_NEG :=, INP_SIM :=, DELAY_TIME :=, DELAY_TIME_OFF :=, INSTANCE := 'DRP-P03.02', RESTART :=, VISIBILITY :=, OPdwCmd :=, QdwState =>, QLOCK =>, QSIM =>, QON =>, QON_DELAY =>, QOFF =>, QOFF_DELAY =>, QOUT =>, QDELAY_TIME =>, QDELAY_TIME_OFF =>, QINP =>, QERR =>, QERR_EXTERN =>, QwAlarm =>)
   END_RUNG
   // the same network as SCL:
   #"DRP-P03.02"(LIOP_SEL := #init, L_RESET := #Reset, INP := "DRP-P03.02", INSTANCE := 'DRP-P03.02');   // "Digital"
END_REGION

REGION Network 6: DRP-P04.01
   RUNG wire#powerrail
      #"DRP-P04.01"(LOCK :=, ERR_EXTERN :=, LIOP_SEL := #init, L_SIM :=, L_RESET := #Reset, INP := "DRP-P04.01", INP_NEG :=, INP_SIM :=, DELAY_TIME :=, DELAY_TIME_OFF :=, INSTANCE := 'DRP-P04.01', RESTART :=, VISIBILITY :=, OPdwCmd :=, QdwState =>, QLOCK =>, QSIM =>, QON =>, QON_DELAY =>, QOFF =>, QOFF_DELAY =>, QOUT =>, QDELAY_TIME =>, QDELAY_TIME_OFF =>, QINP =>, QERR =>, QERR_EXTERN =>, QwAlarm =>)
   END_RUNG
   // the same network as SCL:
   #"DRP-P04.01"(LIOP_SEL := #init, L_RESET := #Reset, INP := "DRP-P04.01", INSTANCE := 'DRP-P04.01');   // "Digital"
END_REGION

REGION Network 7: DRP-P05.01
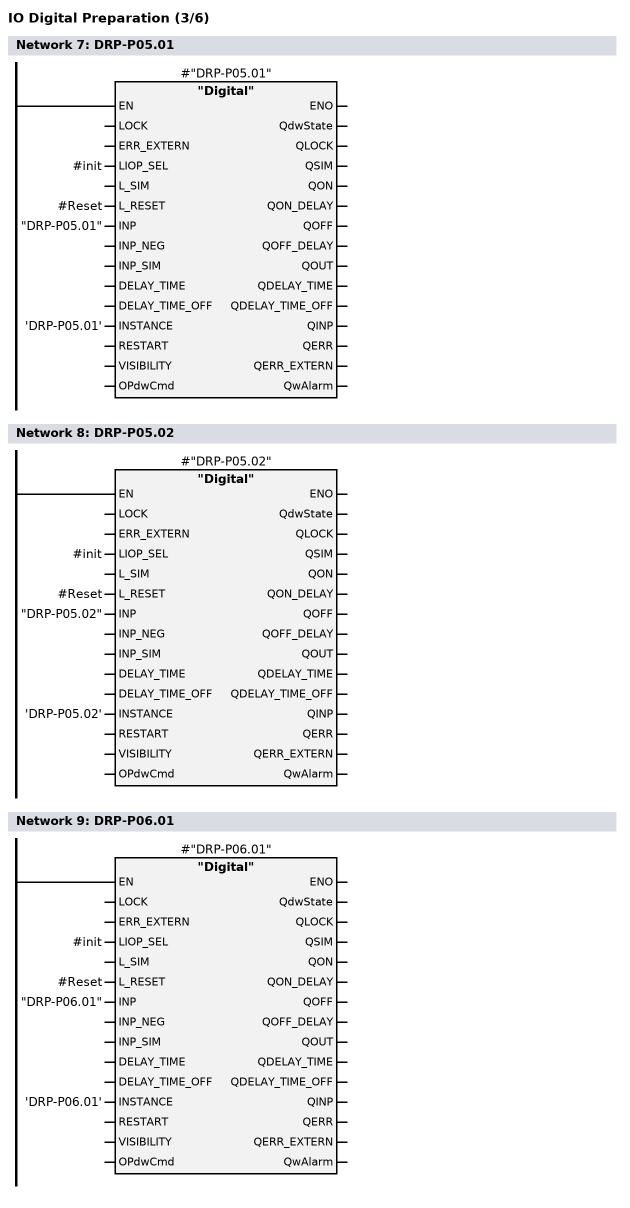
   RUNG wire#powerrail
      #"DRP-P05.01"(LOCK :=, ERR_EXTERN :=, LIOP_SEL := #init, L_SIM :=, L_RESET := #Reset, INP := "DRP-P05.01", INP_NEG :=, INP_SIM :=, DELAY_TIME :=, DELAY_TIME_OFF :=, INSTANCE := 'DRP-P05.01', RESTART :=, VISIBILITY :=, OPdwCmd :=, QdwState =>, QLOCK =>, QSIM =>, QON =>, QON_DELAY =>, QOFF =>, QOFF_DELAY =>, QOUT =>, QDELAY_TIME =>, QDELAY_TIME_OFF =>, QINP =>, QERR =>, QERR_EXTERN =>, QwAlarm =>)
   END_RUNG
   // the same network as SCL:
   #"DRP-P05.01"(LIOP_SEL := #init, L_RESET := #Reset, INP := "DRP-P05.01", INSTANCE := 'DRP-P05.01');   // "Digital"
END_REGION

REGION Network 8: DRP-P05.02
   RUNG wire#powerrail
      #"DRP-P05.02"(LOCK :=, ERR_EXTERN :=, LIOP_SEL := #init, L_SIM :=, L_RESET := #Reset, INP := "DRP-P05.02", INP_NEG :=, INP_SIM :=, DELAY_TIME :=, DELAY_TIME_OFF :=, INSTANCE := 'DRP-P05.02', RESTART :=, VISIBILITY :=, OPdwCmd :=, QdwState =>, QLOCK =>, QSIM =>, QON =>, QON_DELAY =>, QOFF =>, QOFF_DELAY =>, QOUT =>, QDELAY_TIME =>, QDELAY_TIME_OFF =>, QINP =>, QERR =>, QERR_EXTERN =>, QwAlarm =>)
   END_RUNG
   // the same network as SCL:
   #"DRP-P05.02"(LIOP_SEL := #init, L_RESET := #Reset, INP := "DRP-P05.02", INSTANCE := 'DRP-P05.02');   // "Digital"
END_REGION

REGION Network 9: DRP-P06.01
   RUNG wire#powerrail
      #"DRP-P06.01"(LOCK :=, ERR_EXTERN :=, LIOP_SEL := #init, L_SIM :=, L_RESET := #Reset, INP := "DRP-P06.01", INP_NEG :=, INP_SIM :=, DELAY_TIME :=, DELAY_TIME_OFF :=, INSTANCE := 'DRP-P06.01', RESTART :=, VISIBILITY :=, OPdwCmd :=, QdwState =>, QLOCK =>, QSIM =>, QON =>, QON_DELAY =>, QOFF =>, QOFF_DELAY =>, QOUT =>, QDELAY_TIME =>, QDELAY_TIME_OFF =>, QINP =>, QERR =>, QERR_EXTERN =>, QwAlarm =>)
   END_RUNG
   // the same network as SCL:
   #"DRP-P06.01"(LIOP_SEL := #init, L_RESET := #Reset, INP := "DRP-P06.01", INSTANCE := 'DRP-P06.01');   // "Digital"
END_REGION

REGION Network 10: DRP-P07.01
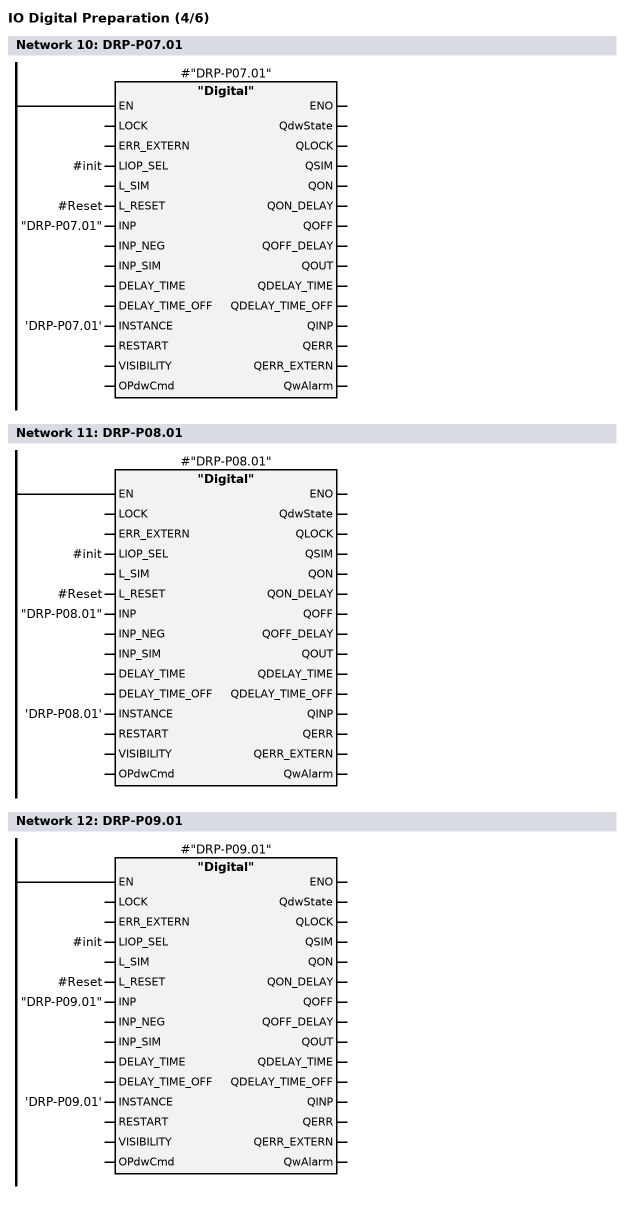
   RUNG wire#powerrail
      #"DRP-P07.01"(LOCK :=, ERR_EXTERN :=, LIOP_SEL := #init, L_SIM :=, L_RESET := #Reset, INP := "DRP-P07.01", INP_NEG :=, INP_SIM :=, DELAY_TIME :=, DELAY_TIME_OFF :=, INSTANCE := 'DRP-P07.01', RESTART :=, VISIBILITY :=, OPdwCmd :=, QdwState =>, QLOCK =>, QSIM =>, QON =>, QON_DELAY =>, QOFF =>, QOFF_DELAY =>, QOUT =>, QDELAY_TIME =>, QDELAY_TIME_OFF =>, QINP =>, QERR =>, QERR_EXTERN =>, QwAlarm =>)
   END_RUNG
   // the same network as SCL:
   #"DRP-P07.01"(LIOP_SEL := #init, L_RESET := #Reset, INP := "DRP-P07.01", INSTANCE := 'DRP-P07.01');   // "Digital"
END_REGION

REGION Network 11: DRP-P08.01
   RUNG wire#powerrail
      #"DRP-P08.01"(LOCK :=, ERR_EXTERN :=, LIOP_SEL := #init, L_SIM :=, L_RESET := #Reset, INP := "DRP-P08.01", INP_NEG :=, INP_SIM :=, DELAY_TIME :=, DELAY_TIME_OFF :=, INSTANCE := 'DRP-P08.01', RESTART :=, VISIBILITY :=, OPdwCmd :=, QdwState =>, QLOCK =>, QSIM =>, QON =>, QON_DELAY =>, QOFF =>, QOFF_DELAY =>, QOUT =>, QDELAY_TIME =>, QDELAY_TIME_OFF =>, QINP =>, QERR =>, QERR_EXTERN =>, QwAlarm =>)
   END_RUNG
   // the same network as SCL:
   #"DRP-P08.01"(LIOP_SEL := #init, L_RESET := #Reset, INP := "DRP-P08.01", INSTANCE := 'DRP-P08.01');   // "Digital"
END_REGION

REGION Network 12: DRP-P09.01
   RUNG wire#powerrail
      #"DRP-P09.01"(LOCK :=, ERR_EXTERN :=, LIOP_SEL := #init, L_SIM :=, L_RESET := #Reset, INP := "DRP-P09.01", INP_NEG :=, INP_SIM :=, DELAY_TIME :=, DELAY_TIME_OFF :=, INSTANCE := 'DRP-P09.01', RESTART :=, VISIBILITY :=, OPdwCmd :=, QdwState =>, QLOCK =>, QSIM =>, QON =>, QON_DELAY =>, QOFF =>, QOFF_DELAY =>, QOUT =>, QDELAY_TIME =>, QDELAY_TIME_OFF =>, QINP =>, QERR =>, QERR_EXTERN =>, QwAlarm =>)
   END_RUNG
   // the same network as SCL:
   #"DRP-P09.01"(LIOP_SEL := #init, L_RESET := #Reset, INP := "DRP-P09.01", INSTANCE := 'DRP-P09.01');   // "Digital"
END_REGION

REGION Network 13: DRP-P09.02
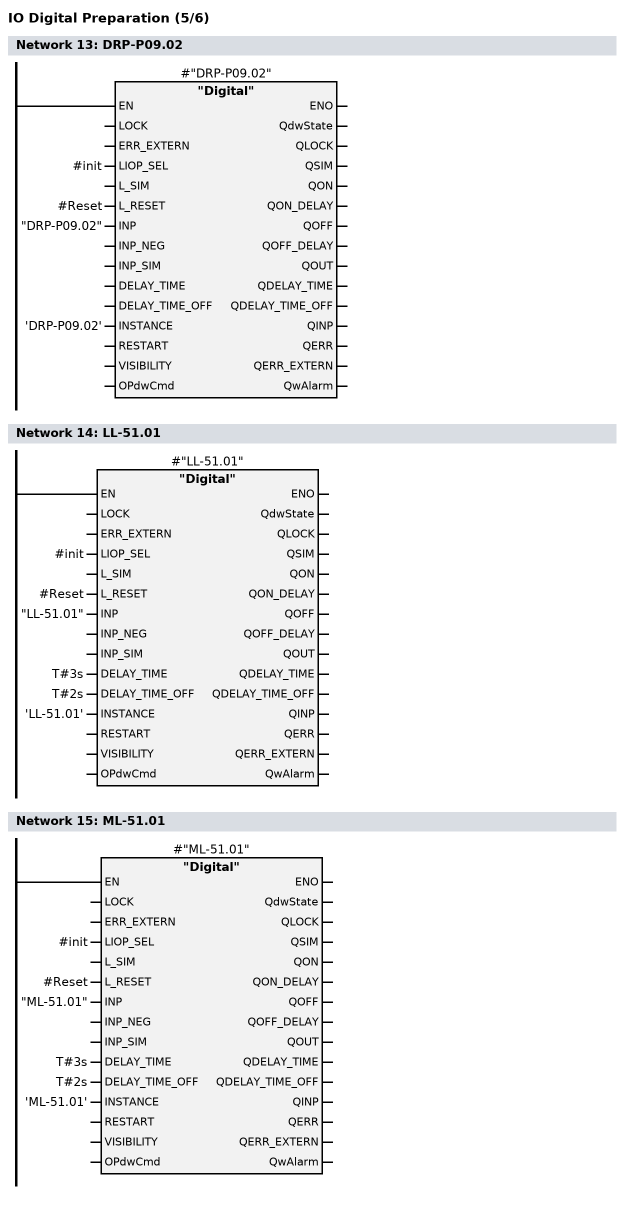
   RUNG wire#powerrail
      #"DRP-P09.02"(LOCK :=, ERR_EXTERN :=, LIOP_SEL := #init, L_SIM :=, L_RESET := #Reset, INP := "DRP-P09.02", INP_NEG :=, INP_SIM :=, DELAY_TIME :=, DELAY_TIME_OFF :=, INSTANCE := 'DRP-P09.02', RESTART :=, VISIBILITY :=, OPdwCmd :=, QdwState =>, QLOCK =>, QSIM =>, QON =>, QON_DELAY =>, QOFF =>, QOFF_DELAY =>, QOUT =>, QDELAY_TIME =>, QDELAY_TIME_OFF =>, QINP =>, QERR =>, QERR_EXTERN =>, QwAlarm =>)
   END_RUNG
   // the same network as SCL:
   #"DRP-P09.02"(LIOP_SEL := #init, L_RESET := #Reset, INP := "DRP-P09.02", INSTANCE := 'DRP-P09.02');   // "Digital"
END_REGION

REGION Network 14: LL-51.01
   RUNG wire#powerrail
      #"LL-51.01"(LOCK :=, ERR_EXTERN :=, LIOP_SEL := #init, L_SIM :=, L_RESET := #Reset, INP := "LL-51.01", INP_NEG :=, INP_SIM :=, DELAY_TIME := T#3s, DELAY_TIME_OFF := T#2s, INSTANCE := 'LL-51.01', RESTART :=, VISIBILITY :=, OPdwCmd :=, QdwState =>, QLOCK =>, QSIM =>, QON =>, QON_DELAY =>, QOFF =>, QOFF_DELAY =>, QOUT =>, QDELAY_TIME =>, QDELAY_TIME_OFF =>, QINP =>, QERR =>, QERR_EXTERN =>, QwAlarm =>)
   END_RUNG
   // the same network as SCL:
   #"LL-51.01"(LIOP_SEL := #init,   // "Digital"
               L_RESET := #Reset,
               INP := "LL-51.01",
               DELAY_TIME := T#3s,
               DELAY_TIME_OFF := T#2s,
               INSTANCE := 'LL-51.01');
END_REGION

REGION Network 15: ML-51.01
   RUNG wire#powerrail
      #"ML-51.01"(LOCK :=, ERR_EXTERN :=, LIOP_SEL := #init, L_SIM :=, L_RESET := #Reset, INP := "ML-51.01", INP_NEG :=, INP_SIM :=, DELAY_TIME := T#3s, DELAY_TIME_OFF := T#2s, INSTANCE := 'ML-51.01', RESTART :=, VISIBILITY :=, OPdwCmd :=, QdwState =>, QLOCK =>, QSIM =>, QON =>, QON_DELAY =>, QOFF =>, QOFF_DELAY =>, QOUT =>, QDELAY_TIME =>, QDELAY_TIME_OFF =>, QINP =>, QERR =>, QERR_EXTERN =>, QwAlarm =>)
   END_RUNG
   // the same network as SCL:
   #"ML-51.01"(LIOP_SEL := #init,   // "Digital"
               L_RESET := #Reset,
               INP := "ML-51.01",
               DELAY_TIME := T#3s,
               DELAY_TIME_OFF := T#2s,
               INSTANCE := 'ML-51.01');
END_REGION

REGION Network 16: HL-51.01
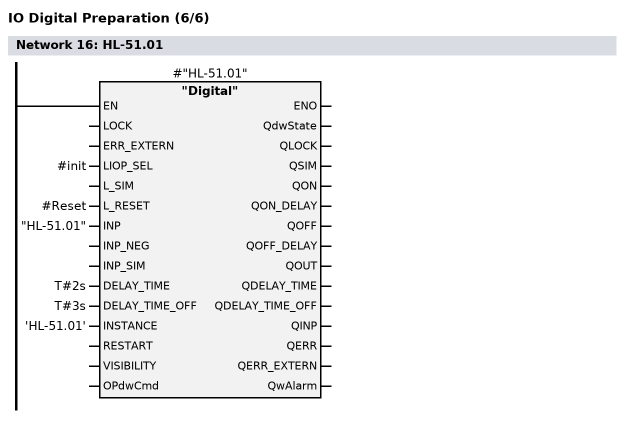
   RUNG wire#powerrail
      #"HL-51.01"(LOCK :=, ERR_EXTERN :=, LIOP_SEL := #init, L_SIM :=, L_RESET := #Reset, INP := "HL-51.01", INP_NEG :=, INP_SIM :=, DELAY_TIME := T#2s, DELAY_TIME_OFF := T#3s, INSTANCE := 'HL-51.01', RESTART :=, VISIBILITY :=, OPdwCmd :=, QdwState =>, QLOCK =>, QSIM =>, QON =>, QON_DELAY =>, QOFF =>, QOFF_DELAY =>, QOUT =>, QDELAY_TIME =>, QDELAY_TIME_OFF =>, QINP =>, QERR =>, QERR_EXTERN =>, QwAlarm =>)
   END_RUNG
   // the same network as SCL:
   #"HL-51.01"(LIOP_SEL := #init,   // "Digital"
               L_RESET := #Reset,
               INP := "HL-51.01",
               DELAY_TIME := T#2s,
               DELAY_TIME_OFF := T#3s,
               INSTANCE := 'HL-51.01');
END_REGION
END_FUNCTION_BLOCK

FUNCTION_BLOCK "BFT_ChiliAwetan"   // FB361, LAD
{ S7_Optimized_Access := 'TRUE' }
VERSION : 0.1
// stored: AutoNumber false, IsIECCheckEnabled false, IsRetainMemResEnabled false, MemoryReserve 100, SetENOAutomatically false, UDAEnableTagReadback false
   VAR_INPUT
      IN_FBAV_Inload : Bool;
      IN_FBAV_Outlet : Bool;
      IN_FBAV_Transfer : Bool;
      IN_FBAV_CIP_Tank : Bool;
      IN_FBAV_CIP_Line : Bool;
      IN_FBP_Inload : Bool;
      IN_FBP_Inload_SP : Real;
      IN_FBP_Transfer : Bool;
      IN_FBP_Transfer_SP : Real;
      IN_FBP_CIP : Bool;
      IN_FBP_CIP_Sp : Real;
      IN_LT01 : Real;
      "LCS Start" : Bool;
      "LCS Stop" : Bool;
      "LCS EMS" : Bool;
      IN_Dose_Run : Bool;
      IN_Dose_Held : Bool;
      IN_Dose_Complete : Bool;
      IN_Dose_Header_1 : Bool;
      IN_Dose_Header_2 : Bool;
      IN_Dose_Valve_Cmd : Bool;
      IN_Dose_Pump_Cmd : Bool;
      IN_Dose_Pump_Sp : Real;
      IN_Dose_LineOK : Bool;
      "Inload Busy" : Bool;
      IN_Prod_Ready : Bool;
      IN_Prod_LineOpen : Bool;
      IN_SupplyOn : Bool;
      IN_Prod_Transfer_Comp : Bool;
      "CIP Pulse" : Bool;
      "CIP Supply ON" : Bool;
      "CIP Req OK" : Bool;
      "CIP Complete" : Bool;
      "CIP Busy" : Bool;
   END_VAR
   VAR_OUTPUT
      Out_AV_Inload : Bool;
      Out_AV_Outlet : Bool;
      Out_AV_Transfer : Bool;
      Out_AV_CIP_Tank : Bool;
      Out_AV_CIP_Line : Bool;
      Out_P_Inload : Bool;
      Out_P_Inload_Sp : Real;
      Out_P_Transfer : Bool;
      Out_P_Transfer_Sp : Real;
      Out_P_CIP : Bool;
      Out_P_CIP_Sp : Real;
      Out_Prod_Req : Bool;
      Out_Prod_LineOpen : Bool;
      Out_CIP_Req : Bool;
      Out_CIP_LineOpen : Bool;
   END_VAR
   VAR
      Cmd : Struct
         Inload : Bool;
         Ready_for_Tranfer : Bool;
         CIP_Tank : Bool;
         CIP_Line : Bool;
      END_STRUCT;
   END_VAR
   VAR RETAIN
      Param : Struct
         SP_Level_LL : Real := 10.0;
         SP_Level_ML : Real := 80.0;
         SP_Level_HL : Real := 100.0;
         SupplyPump_SP_Speed : Real := 80.0;
         L_Hi_Lim : Real := 100.0;
         L_Lo_Lim : Real := 0.0;
         L_Hys : Real := 2.0;
         FlushingTime : DInt := 10000;
         CIP_Trf_SP_Speed : Real := 80.0;
         CIP_Ret_ON_SP : Real := 5.0;
         CIP_Ret_OFF_SP : Real;
      END_STRUCT;
   END_VAR
   VAR
      State : Struct   // Tank in loading state
         Tank_LL : Bool;
         Tank_ML : Bool;
         Tank_HL : Bool;
         Tank_inCIP : Bool;
         Tank_CIP_Enable : Bool;
         Line_inCIP : Bool;
         Line_CIP_Enable : Bool;
         CIP_Return_On : Bool;
         Inloading : Bool;
         Inload_Enable : Bool;
         Ready_For_Transfer : Bool;
         Ready_For_Transfer_Ena : Bool;
         Tank_Available : Bool;
         Transfer_On_Prog : Bool;
      END_STRUCT;
      alwaysON : Bool;
      L_Hys_Abs : Real;
      Hys_Level_HL : Real;
      Hys_Level_ML : Real;
      Hys_Level_LL : Real;
      r : Struct
         PosE1 : Bool;
         PosE2 : Bool;
         PosE3 : Bool;
         PosE4 : Bool;
         PosE5 : Bool;
         PosE6 : Bool;
         PosE7 : Bool;
         PosE8 : Bool;
         PosE9 : Bool;
         PosE10 : Bool;
         PosE11 : Bool;
         PosE12 : Bool;
         PosE13 : Bool;
         PosE14 : Bool;
         PosE15 : Bool;
         PosE16 : Bool;
         PosE17 : Bool;
         PosE18 : Bool;
         PosE19 : Bool;
         PosE20 : Bool;
         PosE21 : Bool;
         PosE22 : Bool;
         PosE23 : Bool;
         PosE24 : Bool;
         PosE25 : Bool;
         PosE26 : Bool;
         PosE27 : Bool;
         PosE28 : Bool;
         PosE29 : Bool;
         PosE30 : Bool;
         PosE31 : Bool;
         PosE32 : Bool;
      END_STRUCT;
      Actuator : Struct
         AV_Inload : Bool;
         AV_Outlet : Bool;
         AV_Transfer : Bool;
         AV_CIP_Tank : Bool;
         AV_CIP_Line : Bool;
         P_Transfer : Bool;
         P_Inload : Bool;
         P_CIP : Bool;
      END_STRUCT;
      FlushingTim : TON_TIME;
      SPumpTim { S7_SetPoint := 'True'} : TON_TIME;
      AVinloadTim { S7_SetPoint := 'True'} : TON_TIME;
      Pump_TF_On_Time { S7_SetPoint := 'True'} : TON_TIME;
   END_VAR
   VAR_TEMP   // added for the SCL form of the ladder/FBD networks
      _w1 : Bool;
      _w2 : Bool;
   END_VAR
BEGIN

REGION Network 1: Always_ON
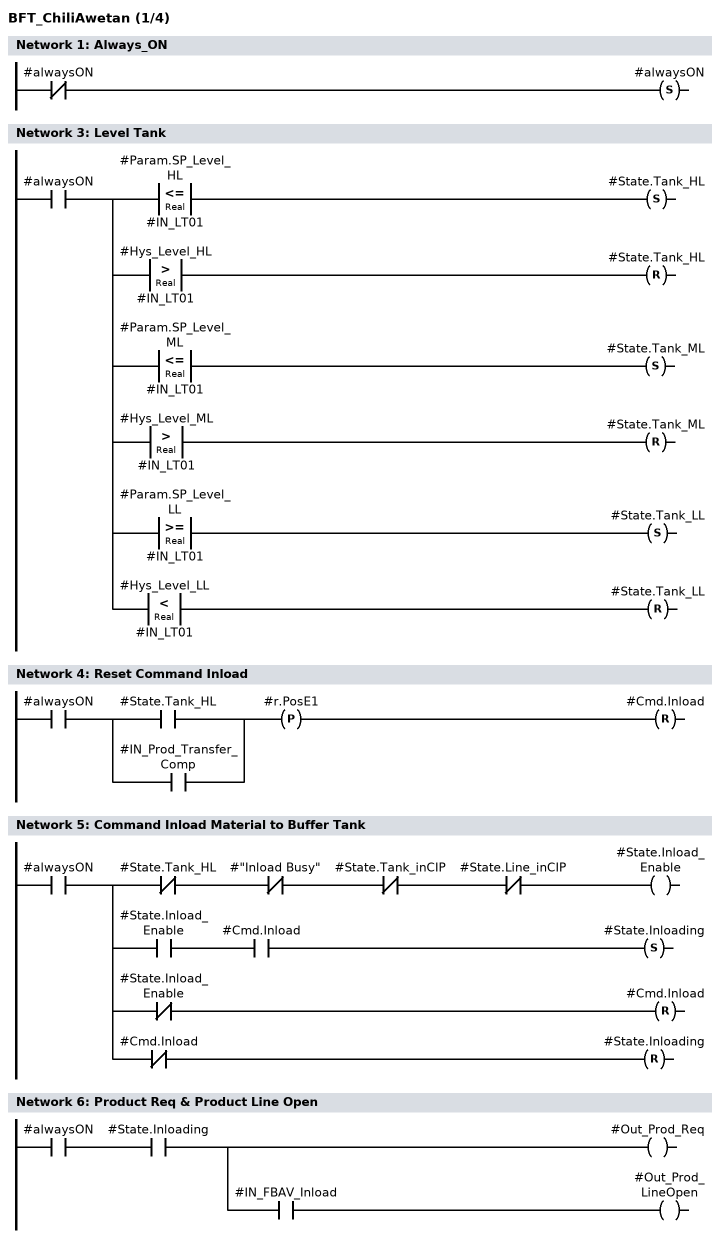
   RUNG wire#powerrail
      I_Contact( #alwaysON )
      S_Coil( #alwaysON )
   END_RUNG
   // the same network as SCL:
   IF NOT #alwaysON THEN #alwaysON := TRUE; END_IF;
END_REGION

NETWORK
TITLE = Hys Calculation
//Level Hys Absolute
      L     #Param.L_Hi_Lim;
      L     #Param.L_Lo_Lim;
      -R;
      L     100.0;
      /R;
      L     #Param.L_Hys;
      *R;
      T     #L_Hys_Abs;
//Tank High Level
      L     #Param.SP_Level_HL;
      L     #L_Hys_Abs;
      -R;
      T     #Hys_Level_HL;
//Tank Mid Level
      L     #Param.SP_Level_ML;
      L     #L_Hys_Abs;
      -R;
      T     #Hys_Level_ML;
//Tank Low Level
      L     #Param.SP_Level_LL;
      L     #L_Hys_Abs;
      +R;
      T     #Hys_Level_LL;


REGION Network 3: Level Tank
   RUNG wire#powerrail
      Contact( #alwaysON )
      wire#w1
      { S7_Templates := "SrcType := Real" } LE_Contact(in1 := #Param.SP_Level_HL, in2 := #IN_LT01)
      S_Coil( #State.Tank_HL )
   END_RUNG
   RUNG wire#w1
      { S7_Templates := "SrcType := Real" } GT_Contact(in1 := #Hys_Level_HL, in2 := #IN_LT01)
      R_Coil( #State.Tank_HL )
   END_RUNG
   RUNG wire#w1
      { S7_Templates := "SrcType := Real" } LE_Contact(in1 := #Param.SP_Level_ML, in2 := #IN_LT01)
      S_Coil( #State.Tank_ML )
   END_RUNG
   RUNG wire#w1
      { S7_Templates := "SrcType := Real" } GT_Contact(in1 := #Hys_Level_ML, in2 := #IN_LT01)
      R_Coil( #State.Tank_ML )
   END_RUNG
   RUNG wire#w1
      { S7_Templates := "SrcType := Real" } GE_Contact(in1 := #Param.SP_Level_LL, in2 := #IN_LT01)
      S_Coil( #State.Tank_LL )
   END_RUNG
   RUNG wire#w1
      { S7_Templates := "SrcType := Real" } LT_Contact(in1 := #Hys_Level_LL, in2 := #IN_LT01)
      R_Coil( #State.Tank_LL )
   END_RUNG
   // the same network as SCL:
   IF #alwaysON AND (#Param.SP_Level_HL <= #IN_LT01) THEN #State.Tank_HL := TRUE; END_IF;
   IF #alwaysON AND (#Hys_Level_HL > #IN_LT01) THEN #State.Tank_HL := FALSE; END_IF;
   IF #alwaysON AND (#Param.SP_Level_ML <= #IN_LT01) THEN #State.Tank_ML := TRUE; END_IF;
   IF #alwaysON AND (#Hys_Level_ML > #IN_LT01) THEN #State.Tank_ML := FALSE; END_IF;
   IF #alwaysON AND (#Param.SP_Level_LL >= #IN_LT01) THEN #State.Tank_LL := TRUE; END_IF;
   IF #alwaysON AND (#Hys_Level_LL < #IN_LT01) THEN #State.Tank_LL := FALSE; END_IF;
END_REGION

REGION Network 4: Reset Command Inload
   RUNG wire#powerrail
      Contact( #alwaysON )
      wire#w1
      Contact( #State.Tank_HL )
      wire#w2
      P_Trig( #r.PosE1 )
      R_Coil( #Cmd.Inload )
   END_RUNG
   RUNG wire#w1
      Contact( #IN_Prod_Transfer_Comp )
   END_RUNG wire#w2
   // the same network as SCL:
   #_w1 := #alwaysON AND (#State.Tank_HL OR #IN_Prod_Transfer_Comp);
   #_w2 := #_w1 AND NOT #r.PosE1;   // rising edge
   #r.PosE1 := #_w1;
   IF #_w2 THEN #Cmd.Inload := FALSE; END_IF;
END_REGION

REGION Network 5: Command Inload Material to Buffer Tank
   RUNG wire#powerrail
      Contact( #alwaysON )
      wire#w1
      I_Contact( #State.Tank_HL )
      I_Contact( #"Inload Busy" )
      I_Contact( #State.Tank_inCIP )
      I_Contact( #State.Line_inCIP )
      Coil( #State.Inload_Enable )
   END_RUNG
   RUNG wire#w1
      Contact( #State.Inload_Enable )
      Contact( #Cmd.Inload )
      S_Coil( #State.Inloading )
   END_RUNG
   RUNG wire#w1
      I_Contact( #State.Inload_Enable )
      R_Coil( #Cmd.Inload )
   END_RUNG
   RUNG wire#w1
      I_Contact( #Cmd.Inload )
      R_Coil( #State.Inloading )
   END_RUNG
   // the same network as SCL:
   #State.Inload_Enable := #alwaysON AND NOT #State.Tank_HL AND NOT #"Inload Busy" AND NOT #State.Tank_inCIP AND NOT #State.Line_inCIP;
   IF #alwaysON AND #State.Inload_Enable AND #Cmd.Inload THEN #State.Inloading := TRUE; END_IF;
   IF #alwaysON AND NOT #State.Inload_Enable THEN #Cmd.Inload := FALSE; END_IF;
   IF #alwaysON AND NOT #Cmd.Inload THEN #State.Inloading := FALSE; END_IF;
END_REGION

REGION Network 6: Product Req & Product Line Open
   RUNG wire#powerrail
      Contact( #alwaysON )
      Contact( #State.Inloading )
      wire#w1
      Coil( #Out_Prod_Req )
   END_RUNG
   RUNG wire#w1
      Contact( #IN_FBAV_Inload )
      Coil( #Out_Prod_LineOpen )
   END_RUNG
   // the same network as SCL:
   #Out_Prod_Req := #alwaysON AND #State.Inloading;
   #Out_Prod_LineOpen := #Out_Prod_Req AND #IN_FBAV_Inload;
END_REGION

REGION Network 8: Tank Ready for Transfer to Blending
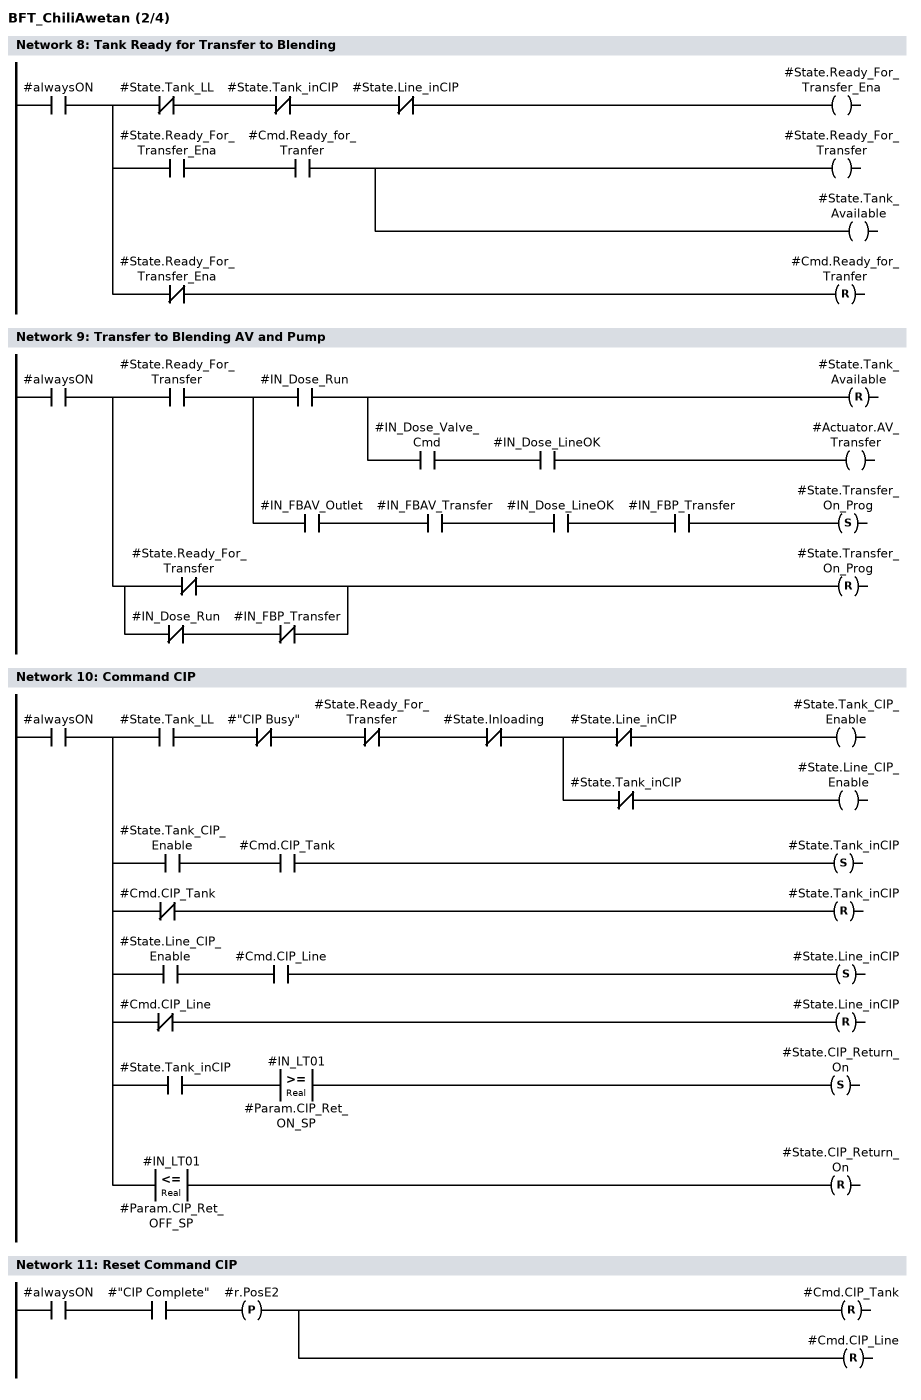
   RUNG wire#powerrail
      Contact( #alwaysON )
      wire#w1
      I_Contact( #State.Tank_LL )
      I_Contact( #State.Tank_inCIP )
      I_Contact( #State.Line_inCIP )
      Coil( #State.Ready_For_Transfer_Ena )
   END_RUNG
   RUNG wire#w1
      Contact( #State.Ready_For_Transfer_Ena )
      Contact( #Cmd.Ready_for_Tranfer )
      wire#w2
      Coil( #State.Ready_For_Transfer )
   END_RUNG
   RUNG wire#w2
      Coil( #State.Tank_Available )
   END_RUNG
   RUNG wire#w1
      I_Contact( #State.Ready_For_Transfer_Ena )
      R_Coil( #Cmd.Ready_for_Tranfer )
   END_RUNG
   // the same network as SCL:
   #State.Ready_For_Transfer_Ena := #alwaysON AND NOT #State.Tank_LL AND NOT #State.Tank_inCIP AND NOT #State.Line_inCIP;
   #State.Ready_For_Transfer := #alwaysON AND #State.Ready_For_Transfer_Ena AND #Cmd.Ready_for_Tranfer;
   #State.Tank_Available := #State.Ready_For_Transfer;
   IF #alwaysON AND NOT #State.Ready_For_Transfer_Ena THEN #Cmd.Ready_for_Tranfer := FALSE; END_IF;
END_REGION

REGION Network 9: Transfer to Blending AV and Pump
   RUNG wire#powerrail
      Contact( #alwaysON )
      wire#w1
      Contact( #State.Ready_For_Transfer )
      wire#w2
      Contact( #IN_Dose_Run )
      wire#w3
      R_Coil( #State.Tank_Available )
   END_RUNG
   RUNG wire#w3
      Contact( #IN_Dose_Valve_Cmd )
      Contact( #IN_Dose_LineOK )
      Coil( #Actuator.AV_Transfer )
   END_RUNG
   RUNG wire#w2
      Contact( #IN_FBAV_Outlet )
      Contact( #IN_FBAV_Transfer )
      Contact( #IN_Dose_LineOK )
      Contact( #IN_FBP_Transfer )
      S_Coil( #State.Transfer_On_Prog )
   END_RUNG
   RUNG wire#w1
      I_Contact( #State.Ready_For_Transfer )
      wire#w4
      R_Coil( #State.Transfer_On_Prog )
   END_RUNG
   RUNG wire#w1
      I_Contact( #IN_Dose_Run )
      I_Contact( #IN_FBP_Transfer )
   END_RUNG wire#w4
   // the same network as SCL:
   #_w1 := #alwaysON AND #State.Ready_For_Transfer;
   #_w2 := #_w1 AND #IN_Dose_Run;
   IF #_w2 THEN #State.Tank_Available := FALSE; END_IF;
   #Actuator.AV_Transfer := #_w2 AND #IN_Dose_Valve_Cmd AND #IN_Dose_LineOK;
   IF #_w1 AND #IN_FBAV_Outlet AND #IN_FBAV_Transfer AND #IN_Dose_LineOK AND #IN_FBP_Transfer THEN
       #State.Transfer_On_Prog := TRUE;
   END_IF;
   IF #alwaysON AND (NOT #State.Ready_For_Transfer OR (NOT #IN_Dose_Run AND NOT #IN_FBP_Transfer)) THEN
       #State.Transfer_On_Prog := FALSE;
   END_IF;
END_REGION

REGION Network 10: Command CIP
   RUNG wire#powerrail
      Contact( #alwaysON )
      wire#w1
      Contact( #State.Tank_LL )
      I_Contact( #"CIP Busy" )
      I_Contact( #State.Ready_For_Transfer )
      I_Contact( #State.Inloading )
      wire#w2
      I_Contact( #State.Line_inCIP )
      Coil( #State.Tank_CIP_Enable )
   END_RUNG
   RUNG wire#w2
      I_Contact( #State.Tank_inCIP )
      Coil( #State.Line_CIP_Enable )
   END_RUNG
   RUNG wire#w1
      Contact( #State.Tank_CIP_Enable )
      Contact( #Cmd.CIP_Tank )
      S_Coil( #State.Tank_inCIP )
   END_RUNG
   RUNG wire#w1
      I_Contact( #Cmd.CIP_Tank )
      R_Coil( #State.Tank_inCIP )
   END_RUNG
   RUNG wire#w1
      Contact( #State.Line_CIP_Enable )
      Contact( #Cmd.CIP_Line )
      S_Coil( #State.Line_inCIP )
   END_RUNG
   RUNG wire#w1
      I_Contact( #Cmd.CIP_Line )
      R_Coil( #State.Line_inCIP )
   END_RUNG
   RUNG wire#w1
      Contact( #State.Tank_inCIP )
      { S7_Templates := "SrcType := Real" } GE_Contact(in1 := #IN_LT01, in2 := #Param.CIP_Ret_ON_SP)
      S_Coil( #State.CIP_Return_On )
   END_RUNG
   RUNG wire#w1
      { S7_Templates := "SrcType := Real" } LE_Contact(in1 := #IN_LT01, in2 := #Param.CIP_Ret_OFF_SP)
      R_Coil( #State.CIP_Return_On )
   END_RUNG
   // the same network as SCL:
   #_w1 := #alwaysON AND #State.Tank_LL AND NOT #"CIP Busy" AND NOT #State.Ready_For_Transfer AND NOT #State.Inloading;
   #State.Tank_CIP_Enable := #_w1 AND NOT #State.Line_inCIP;
   #State.Line_CIP_Enable := #_w1 AND NOT #State.Tank_inCIP;
   IF #alwaysON AND #State.Tank_CIP_Enable AND #Cmd.CIP_Tank THEN #State.Tank_inCIP := TRUE; END_IF;
   IF #alwaysON AND NOT #Cmd.CIP_Tank THEN #State.Tank_inCIP := FALSE; END_IF;
   IF #alwaysON AND #State.Line_CIP_Enable AND #Cmd.CIP_Line THEN #State.Line_inCIP := TRUE; END_IF;
   IF #alwaysON AND NOT #Cmd.CIP_Line THEN #State.Line_inCIP := FALSE; END_IF;
   IF #alwaysON AND #State.Tank_inCIP AND (#IN_LT01 >= #Param.CIP_Ret_ON_SP) THEN
       #State.CIP_Return_On := TRUE;
   END_IF;
   IF #alwaysON AND (#IN_LT01 <= #Param.CIP_Ret_OFF_SP) THEN #State.CIP_Return_On := FALSE; END_IF;
END_REGION

REGION Network 11: Reset Command CIP
   RUNG wire#powerrail
      Contact( #alwaysON )
      Contact( #"CIP Complete" )
      P_Trig( #r.PosE2 )
      wire#w1
      R_Coil( #Cmd.CIP_Tank )
   END_RUNG
   RUNG wire#w1
      R_Coil( #Cmd.CIP_Line )
   END_RUNG
   // the same network as SCL:
   #_w1 := #alwaysON AND #"CIP Complete";
   #_w2 := #_w1 AND NOT #r.PosE2;   // rising edge
   #r.PosE2 := #_w1;
   IF #_w2 THEN
       #Cmd.CIP_Tank := FALSE;
       #Cmd.CIP_Line := FALSE;
   END_IF;
END_REGION

REGION Network 12: CIP Request and CIP Line Open
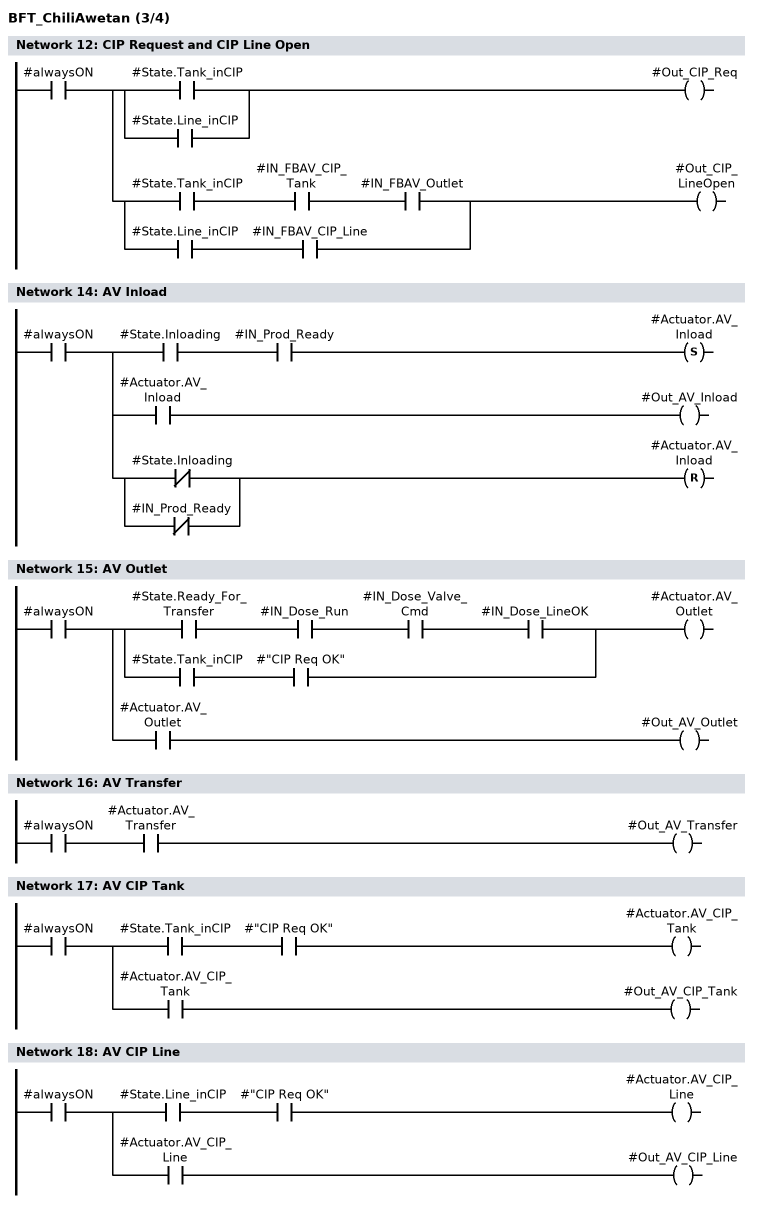
   RUNG wire#powerrail
      Contact( #alwaysON )
      wire#w1
      Contact( #State.Tank_inCIP )
      wire#w2
      Coil( #Out_CIP_Req )
   END_RUNG
   RUNG wire#w1
      Contact( #State.Line_inCIP )
   END_RUNG wire#w2
   RUNG wire#w1
      Contact( #State.Tank_inCIP )
      Contact( #IN_FBAV_CIP_Tank )
      Contact( #IN_FBAV_Outlet )
      wire#w3
      Coil( #Out_CIP_LineOpen )
   END_RUNG
   RUNG wire#w1
      Contact( #State.Line_inCIP )
      Contact( #IN_FBAV_CIP_Line )
   END_RUNG wire#w3
   // the same network as SCL:
   #Out_CIP_Req := #alwaysON AND (#State.Tank_inCIP OR #State.Line_inCIP);
   #Out_CIP_LineOpen := #alwaysON AND ((#State.Tank_inCIP AND #IN_FBAV_CIP_Tank AND #IN_FBAV_Outlet) OR (#State.Line_inCIP AND #IN_FBAV_CIP_Line));
END_REGION

REGION Network 14: AV Inload
   RUNG wire#powerrail
      Contact( #alwaysON )
      wire#w1
      Contact( #State.Inloading )
      Contact( #IN_Prod_Ready )
      S_Coil( #Actuator.AV_Inload )
   END_RUNG
   RUNG wire#w1
      Contact( #Actuator.AV_Inload )
      Coil( #Out_AV_Inload )
   END_RUNG
   RUNG wire#w1
      I_Contact( #State.Inloading )
      wire#w2
      R_Coil( #Actuator.AV_Inload )
   END_RUNG
   RUNG wire#w1
      I_Contact( #IN_Prod_Ready )
   END_RUNG wire#w2
   // the same network as SCL:
   IF #alwaysON AND #State.Inloading AND #IN_Prod_Ready THEN #Actuator.AV_Inload := TRUE; END_IF;
   #Out_AV_Inload := #alwaysON AND #Actuator.AV_Inload;
   IF #alwaysON AND (NOT #State.Inloading OR NOT #IN_Prod_Ready) THEN #Actuator.AV_Inload := FALSE; END_IF;
END_REGION

REGION Network 15: AV Outlet
   RUNG wire#powerrail
      Contact( #alwaysON )
      wire#w1
      Contact( #State.Ready_For_Transfer )
      Contact( #IN_Dose_Run )
      Contact( #IN_Dose_Valve_Cmd )
      Contact( #IN_Dose_LineOK )
      wire#w2
      Coil( #Actuator.AV_Outlet )
   END_RUNG
   RUNG wire#w1
      Contact( #State.Tank_inCIP )
      Contact( #"CIP Req OK" )
   END_RUNG wire#w2
   RUNG wire#w1
      Contact( #Actuator.AV_Outlet )
      Coil( #Out_AV_Outlet )
   END_RUNG
   // the same network as SCL:
   #Actuator.AV_Outlet := #alwaysON AND ((#State.Ready_For_Transfer AND #IN_Dose_Run AND #IN_Dose_Valve_Cmd AND #IN_Dose_LineOK) OR (#State.Tank_inCIP AND #"CIP Req OK"));
   #Out_AV_Outlet := #alwaysON AND #Actuator.AV_Outlet;
END_REGION

REGION Network 16: AV Transfer
   RUNG wire#powerrail
      Contact( #alwaysON )
      Contact( #Actuator.AV_Transfer )
      Coil( #Out_AV_Transfer )
   END_RUNG
   // the same network as SCL:
   #Out_AV_Transfer := #alwaysON AND #Actuator.AV_Transfer;
END_REGION

REGION Network 17: AV CIP Tank
   RUNG wire#powerrail
      Contact( #alwaysON )
      wire#w1
      Contact( #State.Tank_inCIP )
      Contact( #"CIP Req OK" )
      Coil( #Actuator.AV_CIP_Tank )
   END_RUNG
   RUNG wire#w1
      Contact( #Actuator.AV_CIP_Tank )
      Coil( #Out_AV_CIP_Tank )
   END_RUNG
   // the same network as SCL:
   #Actuator.AV_CIP_Tank := #alwaysON AND #State.Tank_inCIP AND #"CIP Req OK";
   #Out_AV_CIP_Tank := #alwaysON AND #Actuator.AV_CIP_Tank;
END_REGION

REGION Network 18: AV CIP Line
   RUNG wire#powerrail
      Contact( #alwaysON )
      wire#w1
      Contact( #State.Line_inCIP )
      Contact( #"CIP Req OK" )
      Coil( #Actuator.AV_CIP_Line )
   END_RUNG
   RUNG wire#w1
      Contact( #Actuator.AV_CIP_Line )
      Coil( #Out_AV_CIP_Line )
   END_RUNG
   // the same network as SCL:
   #Actuator.AV_CIP_Line := #alwaysON AND #State.Line_inCIP AND #"CIP Req OK";
   #Out_AV_CIP_Line := #alwaysON AND #Actuator.AV_CIP_Line;
END_REGION

REGION Network 20: Pump Inload
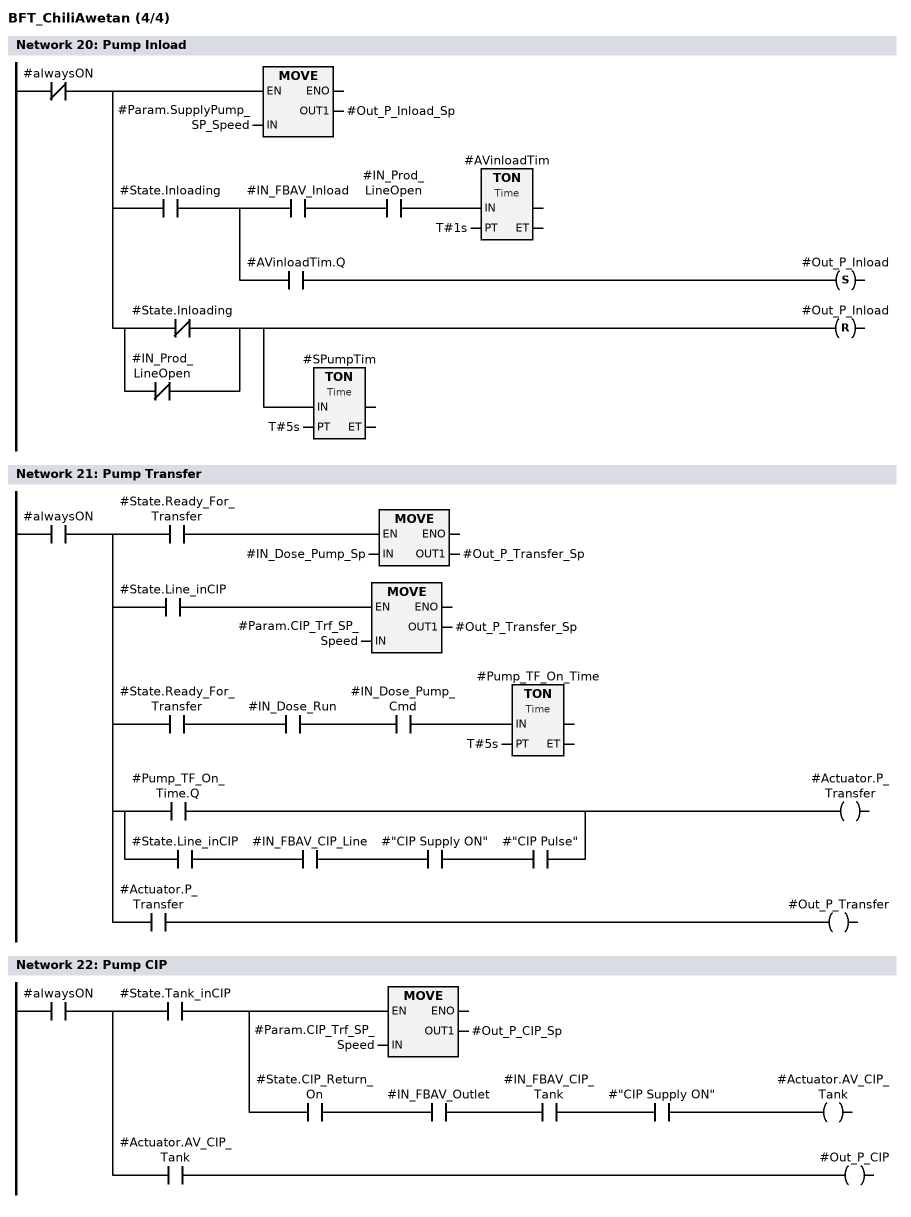
   RUNG wire#powerrail
      I_Contact( #alwaysON )
      wire#w1
      Move(in := #Param.SupplyPump_SP_Speed, out1 => #Out_P_Inload_Sp)
   END_RUNG
   RUNG wire#w1
      Contact( #State.Inloading )
      wire#w2
      Contact( #IN_FBAV_Inload )
      Contact( #IN_Prod_LineOpen )
      { S7_Templates := "time_type := Time" } #AVinloadTim.TON(pt := T#1s, et =>)
   END_RUNG
   RUNG wire#w2
      Contact( #AVinloadTim.Q )
      S_Coil( #Out_P_Inload )
   END_RUNG
   RUNG wire#w1
      I_Contact( #State.Inloading )
      wire#w3
      R_Coil( #Out_P_Inload )
   END_RUNG
   RUNG wire#w1
      I_Contact( #IN_Prod_LineOpen )
   END_RUNG wire#w3
   RUNG wire#w3
      { S7_Templates := "time_type := Time" } #SPumpTim.TON(pt := T#5s, et =>)
   END_RUNG
   // the same network as SCL:
   IF NOT #alwaysON THEN #Out_P_Inload_Sp := #Param.SupplyPump_SP_Speed; END_IF;
   #_w1 := NOT #alwaysON AND #State.Inloading;
   #AVinloadTim(IN := #_w1 AND #IN_FBAV_Inload AND #IN_Prod_LineOpen, PT := T#1s);   // TON
   IF #_w1 AND #AVinloadTim.Q THEN #Out_P_Inload := TRUE; END_IF;
   #_w2 := NOT #alwaysON AND (NOT #State.Inloading OR NOT #IN_Prod_LineOpen);
   IF #_w2 THEN #Out_P_Inload := FALSE; END_IF;
   #SPumpTim(IN := #_w2, PT := T#5s);   // TON
END_REGION

REGION Network 21: Pump Transfer
   RUNG wire#powerrail
      Contact( #alwaysON )
      wire#w1
      Contact( #State.Ready_For_Transfer )
      Move(in := #IN_Dose_Pump_Sp, out1 => #Out_P_Transfer_Sp)
   END_RUNG
   RUNG wire#w1
      Contact( #State.Line_inCIP )
      Move(in := #Param.CIP_Trf_SP_Speed, out1 => #Out_P_Transfer_Sp)
   END_RUNG
   RUNG wire#w1
      Contact( #State.Ready_For_Transfer )
      Contact( #IN_Dose_Run )
      Contact( #IN_Dose_Pump_Cmd )
      { S7_Templates := "time_type := Time" } #Pump_TF_On_Time.TON(pt := T#5s, et =>)
   END_RUNG
   RUNG wire#w1
      Contact( #Pump_TF_On_Time.Q )
      wire#w2
      Coil( #Actuator.P_Transfer )
   END_RUNG
   RUNG wire#w1
      Contact( #State.Line_inCIP )
      Contact( #IN_FBAV_CIP_Line )
      Contact( #"CIP Supply ON" )
      Contact( #"CIP Pulse" )
   END_RUNG wire#w2
   RUNG wire#w1
      Contact( #Actuator.P_Transfer )
      Coil( #Out_P_Transfer )
   END_RUNG
   // the same network as SCL:
   IF #alwaysON AND #State.Ready_For_Transfer THEN #Out_P_Transfer_Sp := #IN_Dose_Pump_Sp; END_IF;
   IF #alwaysON AND #State.Line_inCIP THEN #Out_P_Transfer_Sp := #Param.CIP_Trf_SP_Speed; END_IF;
   #Pump_TF_On_Time(IN := #alwaysON AND #State.Ready_For_Transfer AND #IN_Dose_Run AND #IN_Dose_Pump_Cmd,   // TON
                    PT := T#5s);
   #Actuator.P_Transfer := #alwaysON AND (#Pump_TF_On_Time.Q OR (#State.Line_inCIP AND #IN_FBAV_CIP_Line AND #"CIP Supply ON" AND #"CIP Pulse"));
   #Out_P_Transfer := #alwaysON AND #Actuator.P_Transfer;
END_REGION

REGION Network 22: Pump CIP
   RUNG wire#powerrail
      Contact( #alwaysON )
      wire#w1
      Contact( #State.Tank_inCIP )
      wire#w2
      Move(in := #Param.CIP_Trf_SP_Speed, out1 => #Out_P_CIP_Sp)
   END_RUNG
   RUNG wire#w2
      Contact( #State.CIP_Return_On )
      Contact( #IN_FBAV_Outlet )
      Contact( #IN_FBAV_CIP_Tank )
      Contact( #"CIP Supply ON" )
      Coil( #Actuator.AV_CIP_Tank )
   END_RUNG
   RUNG wire#w1
      Contact( #Actuator.AV_CIP_Tank )
      Coil( #Out_P_CIP )
   END_RUNG
   // the same network as SCL:
   #_w1 := #alwaysON AND #State.Tank_inCIP;
   IF #_w1 THEN #Out_P_CIP_Sp := #Param.CIP_Trf_SP_Speed; END_IF;
   #Actuator.AV_CIP_Tank := #_w1 AND #State.CIP_Return_On AND #IN_FBAV_Outlet AND #IN_FBAV_CIP_Tank AND #"CIP Supply ON";
   #Out_P_CIP := #alwaysON AND #Actuator.AV_CIP_Tank;
END_REGION
END_FUNCTION_BLOCK

FUNCTION_BLOCK "BFT_Tomato"   // FB365, LAD
{ S7_Optimized_Access := 'TRUE' }
VERSION : 0.1
// stored: AutoNumber false, IsIECCheckEnabled false, IsRetainMemResEnabled false, MemoryReserve 100, SetENOAutomatically false, UDAEnableTagReadback false
   VAR_INPUT
      IN_FBAV_Inload : Bool;
      IN_FBAV_Outlet : Bool;
      IN_FBAV_Transfer : Bool;
      IN_FBAV_CIP_Tank : Bool;
      IN_FBAV_CIP_Line : Bool;
      IN_FBAV_Vinegar : Bool;
      IN_FBAV_ProWater : Bool;
      IN_FBP_Inload : Bool;
      IN_FBP_Inload_SP : Real;
      IN_FBP_Transfer : Bool;
      IN_FBP_Transfer_SP : Real;
      IN_FBP_CIP : Bool;
      IN_FBP_CIP_Sp : Real;
      IN_LT01 : Real;
      "LCS Start" : Bool;
      "LCS Stop" : Bool;
      "LCS EMS" : Bool;
      IN_Dose_Run : Bool;
      IN_Dose_Held : Bool;
      IN_Dose_Complete : Bool;
      IN_Dose_Header_1 : Bool;
      IN_Dose_Header_2 : Bool;
      IN_Dose_Valve_Cmd : Bool;
      IN_Dose_Pump_Cmd : Bool;
      IN_Dose_Pump_Sp : Real;
      IN_Dose_LineOK : Bool;
      "Inload Busy" : Bool;
      "CIP Pulse" : Bool;
      "CIP Supply ON" : Bool;
      "CIP Req OK" : Bool;
      "CIP Complete" : Bool;
      "CIP Busy" : Bool;
      "Vinegar Available" : Bool;
      "Vinegar Tank Ready" : Bool;
      "Vinegar Prod Ready" : Bool;
      "Vinegar Valve Open" : Bool;
      "Vinegar Pump Run" : Bool;
      IN_FT_Vinegar : Real;
      ProWater_Req_OK : Bool;
      IN_LDT : Date_And_Time;
   END_VAR
   VAR_OUTPUT
      Out_AV_Inload : Bool;
      Out_AV_Outlet : Bool;
      Out_AV_Transfer : Bool;
      Out_AV_CIP_Tank : Bool;
      Out_AV_CIP_Line : Bool;
      Out_AV_Vinegar : Bool;
      Out_AV_ProWater : Bool;
      Out_P_Inload : Bool;
      Out_P_Inload_Sp : Real;
      Out_P_Transfer : Bool;
      Out_P_Transfer_Sp : Real;
      Out_P_CIP : Bool;
      Out_P_CIP_Sp : Real;
      Out_XA : Bool;
      Out_XA_Speed : Real;
      "Vinegar Req" : Bool;
      ProWater_Req : Bool;
      Out_CIP_Req : Bool;
      Out_CIP_LineOpen : Bool;
   END_VAR
   VAR
      Cmd : Struct
         Inload_Tomato : Bool;
         Inload_ProWater : Bool;
         Ready_for_Tranfer : Bool;
         CIP_Tank : Bool;
         CIP_Line : Bool;
         Agitator_SpeedMode : Bool;
         Agitator_Mode : Bool;
         Agitator_Man_OnOff : Bool;
      END_STRUCT;
   END_VAR
   VAR RETAIN
      Param : Struct
         SP_Level_LL : Real := 10.0;
         SP_Level_ML : Real := 80.0;
         SP_Level_HL : Real := 100.0;
         SP_Level_Agi_ON1 : Real := 20.0;
         SP_Level_Agi_OFF1 : Real := 60.0;
         SP_Level_Agi_ON2 : Real := 62.0;
         SP_Level_Agi_OFF2 : Real := 80.0;
         SP_Level_Agi_ON3 : Real := 82.0;
         Agitator_SP_Speed : Real := 50.0;
         SupplyPump_SP_Speed : Real := 80.0;
         L_Hi_Lim : Real := 100.0;
         L_Lo_Lim : Real := 0.0;
         L_Hys : Real := 2.0;
         FlushingTime : DInt := 10000;
         CIP_Trf_SP_Speed : Real := 80.0;
         CIP_Ret_ON_SP : Real := 5.0;
         CIP_Ret_OFF_SP : Real;
      END_STRUCT;
   END_VAR
   VAR
      State : Struct   // Tank in loading state
         Tank_LL : Bool;
         Tank_ML : Bool;
         Tank_HL : Bool;
         Tank_inCIP : Bool;
         Tank_CIP_Enable : Bool;
         Line_inCIP : Bool;
         Line_CIP_Enable : Bool;
         CIP_Return_On : Bool;
         Inloading : Bool;
         Inload_Enable : Bool;
         Ready_For_Transfer : Bool;
         Ready_For_Transfer_Ena : Bool;
         Tank_Available : Bool;
         Transfer_On_Prog : Bool;
         L_Agi_ON1 : Bool;
         L_Agi_ON2 : Bool;
         L_Agi_ON3 : Bool;
         "Dose EN" : Bool;
         Inloading_ProWater : Bool;
         Inloading_Tomato : Bool;
      END_STRUCT;
      Dose : Struct
         Dose_Start : DWord;
         Dose_Pause : DWord;
         Dose_Stop : DWord;
         Dose_State : DWord;
      END_STRUCT;
      alwaysON : Bool;
      L_Hys_Abs : Real;
      Hys_Level_HL : Real;
      Hys_Level_ML : Real;
      Hys_Level_LL : Real;
      Hys_Level_Agi : Real;
      r : Struct
         PosE1 : Bool;
         PosE2 : Bool;
         PosE3 : Bool;
         PosE4 : Bool;
         PosE5 : Bool;
         PosE6 : Bool;
         PosE7 : Bool;
         PosE8 : Bool;
         PosE9 : Bool;
         PosE10 : Bool;
         PosE11 : Bool;
         PosE12 : Bool;
         PosE13 : Bool;
         PosE14 : Bool;
         PosE15 : Bool;
         PosE16 : Bool;
         PosE17 : Bool;
         PosE18 : Bool;
         PosE19 : Bool;
         PosE20 : Bool;
         PosE21 : Bool;
         PosE22 : Bool;
         PosE23 : Bool;
         PosE24 : Bool;
         PosE25 : Bool;
         PosE26 : Bool;
         PosE27 : Bool;
         PosE28 : Bool;
         PosE29 : Bool;
         PosE30 : Bool;
         PosE31 : Bool;
         PosE32 : Bool;
      END_STRUCT;
      Actuator : Struct
         AV_Inload_Tomato : Bool;
         AV_Inload_ProWater : Bool;
         AV_Outlet : Bool;
         AV_Transfer : Bool;
         AV_CIP_Tank : Bool;
         AV_CIP_Line : Bool;
         P_Transfer : Bool;
         P_Inload : Bool;
         P_CIP : Bool;
         Agitator_level : Bool;
         LCS_OnOff : Bool;
      END_STRUCT;
      FlushingTim : TON_TIME;
      SPumpTim { S7_SetPoint := 'True'} : TON_TIME;
      AVinloadTim { S7_SetPoint := 'True'} : TON_TIME;
      L_AgiTim { S7_SetPoint := 'True'} : TON_TIME;
      SP_Vinegar { S7_SetPoint := 'True'} : "RawDose";
      Dose_Vinegar { S7_SetPoint := 'True'} : "DOSE";
      Vinegar_Ready_State { S7_SetPoint := 'True'} : Bool;
      Vinegar_EN : Bool;
      Pump_TF_On_Time { S7_SetPoint := 'True'} : TON_TIME;
   END_VAR
   VAR_TEMP   // added for the SCL form of the ladder/FBD networks
      _w1 : Bool;
      _w2 : Bool;
   END_VAR
BEGIN

REGION Network 1: Always_ON
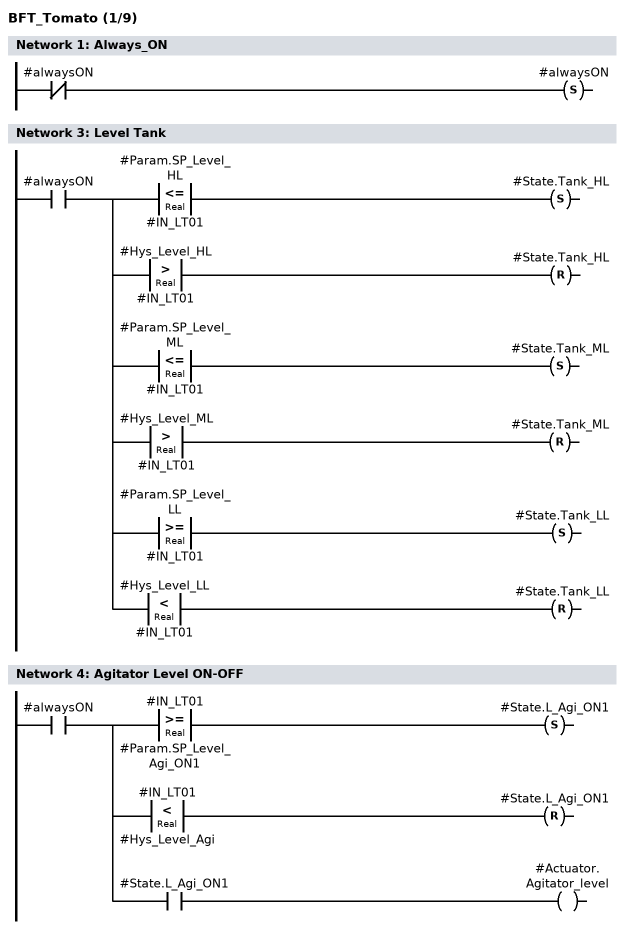
   RUNG wire#powerrail
      I_Contact( #alwaysON )
      S_Coil( #alwaysON )
   END_RUNG
   // the same network as SCL:
   IF NOT #alwaysON THEN #alwaysON := TRUE; END_IF;
END_REGION

NETWORK
TITLE = Hys Calculation
//Level Hys Absolute
      L     #Param.L_Hi_Lim;
      L     #Param.L_Lo_Lim;
      -R;
      L     100.0;
      /R;
      L     #Param.L_Hys;
      *R;
      T     #L_Hys_Abs;
//Tank High Level
      L     #Param.SP_Level_HL;
      L     #L_Hys_Abs;
      -R;
      T     #Hys_Level_HL;
//Tank Mid Level
      L     #Param.SP_Level_ML;
      L     #L_Hys_Abs;
      -R;
      T     #Hys_Level_ML;
//Tank Low Level
      L     #Param.SP_Level_LL;
      L     #L_Hys_Abs;
      +R;
      T     #Hys_Level_LL;
//Level Agi
      L     #Param.SP_Level_Agi_ON1;
      L     #L_Hys_Abs;
      -R;
      T     #Hys_Level_Agi;



REGION Network 3: Level Tank
   RUNG wire#powerrail
      Contact( #alwaysON )
      wire#w1
      { S7_Templates := "SrcType := Real" } LE_Contact(in1 := #Param.SP_Level_HL, in2 := #IN_LT01)
      S_Coil( #State.Tank_HL )
   END_RUNG
   RUNG wire#w1
      { S7_Templates := "SrcType := Real" } GT_Contact(in1 := #Hys_Level_HL, in2 := #IN_LT01)
      R_Coil( #State.Tank_HL )
   END_RUNG
   RUNG wire#w1
      { S7_Templates := "SrcType := Real" } LE_Contact(in1 := #Param.SP_Level_ML, in2 := #IN_LT01)
      S_Coil( #State.Tank_ML )
   END_RUNG
   RUNG wire#w1
      { S7_Templates := "SrcType := Real" } GT_Contact(in1 := #Hys_Level_ML, in2 := #IN_LT01)
      R_Coil( #State.Tank_ML )
   END_RUNG
   RUNG wire#w1
      { S7_Templates := "SrcType := Real" } GE_Contact(in1 := #Param.SP_Level_LL, in2 := #IN_LT01)
      S_Coil( #State.Tank_LL )
   END_RUNG
   RUNG wire#w1
      { S7_Templates := "SrcType := Real" } LT_Contact(in1 := #Hys_Level_LL, in2 := #IN_LT01)
      R_Coil( #State.Tank_LL )
   END_RUNG
   // the same network as SCL:
   IF #alwaysON AND (#Param.SP_Level_HL <= #IN_LT01) THEN #State.Tank_HL := TRUE; END_IF;
   IF #alwaysON AND (#Hys_Level_HL > #IN_LT01) THEN #State.Tank_HL := FALSE; END_IF;
   IF #alwaysON AND (#Param.SP_Level_ML <= #IN_LT01) THEN #State.Tank_ML := TRUE; END_IF;
   IF #alwaysON AND (#Hys_Level_ML > #IN_LT01) THEN #State.Tank_ML := FALSE; END_IF;
   IF #alwaysON AND (#Param.SP_Level_LL >= #IN_LT01) THEN #State.Tank_LL := TRUE; END_IF;
   IF #alwaysON AND (#Hys_Level_LL < #IN_LT01) THEN #State.Tank_LL := FALSE; END_IF;
END_REGION

REGION Network 4: Agitator Level ON-OFF
   RUNG wire#powerrail
      Contact( #alwaysON )
      wire#w1
      { S7_Templates := "SrcType := Real" } GE_Contact(in1 := #IN_LT01, in2 := #Param.SP_Level_Agi_ON1)
      S_Coil( #State.L_Agi_ON1 )
   END_RUNG
   RUNG wire#w1
      { S7_Templates := "SrcType := Real" } LT_Contact(in1 := #IN_LT01, in2 := #Hys_Level_Agi)
      R_Coil( #State.L_Agi_ON1 )
   END_RUNG
   RUNG wire#w1
      Contact( #State.L_Agi_ON1 )
      Coil( #Actuator.Agitator_level )
   END_RUNG
   // the same network as SCL:
   IF #alwaysON AND (#IN_LT01 >= #Param.SP_Level_Agi_ON1) THEN #State.L_Agi_ON1 := TRUE; END_IF;
   IF #alwaysON AND (#IN_LT01 < #Hys_Level_Agi) THEN #State.L_Agi_ON1 := FALSE; END_IF;
   #Actuator.Agitator_level := #alwaysON AND #State.L_Agi_ON1;
END_REGION

REGION Network 5: Agitator
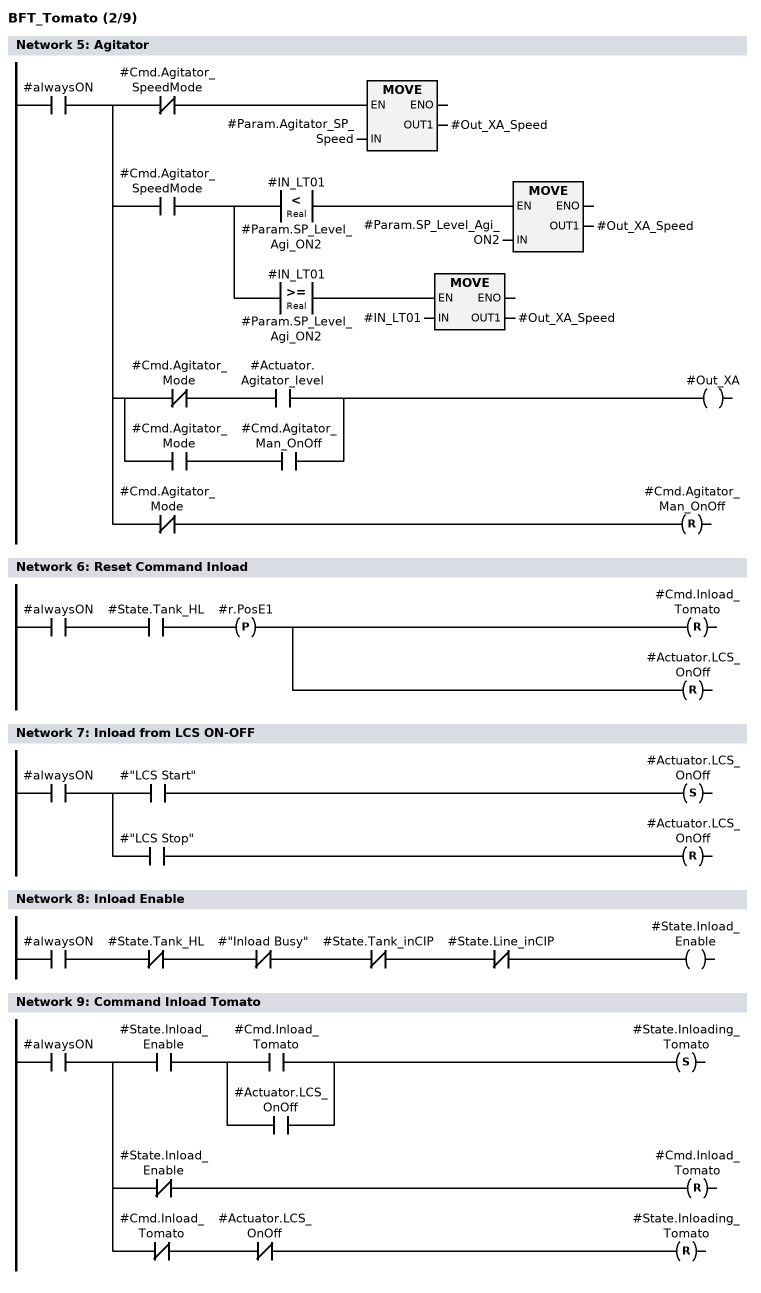
   RUNG wire#powerrail
      Contact( #alwaysON )
      wire#w1
      I_Contact( #Cmd.Agitator_SpeedMode )
      Move(in := #Param.Agitator_SP_Speed, out1 => #Out_XA_Speed)
   END_RUNG
   RUNG wire#w1
      Contact( #Cmd.Agitator_SpeedMode )
      wire#w2
      { S7_Templates := "SrcType := Real" } LT_Contact(in1 := #IN_LT01, in2 := #Param.SP_Level_Agi_ON2)
      Move(in := #Param.SP_Level_Agi_ON2, out1 => #Out_XA_Speed)
   END_RUNG
   RUNG wire#w2
      { S7_Templates := "SrcType := Real" } GE_Contact(in1 := #IN_LT01, in2 := #Param.SP_Level_Agi_ON2)
      Move(in := #IN_LT01, out1 => #Out_XA_Speed)
   END_RUNG
   RUNG wire#w1
      I_Contact( #Cmd.Agitator_Mode )
      Contact( #Actuator.Agitator_level )
      wire#w3
      Coil( #Out_XA )
   END_RUNG
   RUNG wire#w1
      Contact( #Cmd.Agitator_Mode )
      Contact( #Cmd.Agitator_Man_OnOff )
   END_RUNG wire#w3
   RUNG wire#w1
      I_Contact( #Cmd.Agitator_Mode )
      R_Coil( #Cmd.Agitator_Man_OnOff )
   END_RUNG
   // the same network as SCL:
   IF #alwaysON AND NOT #Cmd.Agitator_SpeedMode THEN #Out_XA_Speed := #Param.Agitator_SP_Speed; END_IF;
   #_w1 := #alwaysON AND #Cmd.Agitator_SpeedMode;
   IF #_w1 AND (#IN_LT01 < #Param.SP_Level_Agi_ON2) THEN #Out_XA_Speed := #Param.SP_Level_Agi_ON2; END_IF;
   IF #_w1 AND (#IN_LT01 >= #Param.SP_Level_Agi_ON2) THEN #Out_XA_Speed := #IN_LT01; END_IF;
   #Out_XA := #alwaysON AND ((NOT #Cmd.Agitator_Mode AND #Actuator.Agitator_level) OR (#Cmd.Agitator_Mode AND #Cmd.Agitator_Man_OnOff));
   IF #alwaysON AND NOT #Cmd.Agitator_Mode THEN #Cmd.Agitator_Man_OnOff := FALSE; END_IF;
END_REGION

REGION Network 6: Reset Command Inload
   RUNG wire#powerrail
      Contact( #alwaysON )
      Contact( #State.Tank_HL )
      P_Trig( #r.PosE1 )
      wire#w1
      R_Coil( #Cmd.Inload_Tomato )
   END_RUNG
   RUNG wire#w1
      R_Coil( #Actuator.LCS_OnOff )
   END_RUNG
   // the same network as SCL:
   #_w1 := #alwaysON AND #State.Tank_HL;
   #_w2 := #_w1 AND NOT #r.PosE1;   // rising edge
   #r.PosE1 := #_w1;
   IF #_w2 THEN
       #Cmd.Inload_Tomato := FALSE;
       #Actuator.LCS_OnOff := FALSE;
   END_IF;
END_REGION

REGION Network 7: Inload from LCS ON-OFF
   RUNG wire#powerrail
      Contact( #alwaysON )
      wire#w1
      Contact( #"LCS Start" )
      S_Coil( #Actuator.LCS_OnOff )
   END_RUNG
   RUNG wire#w1
      Contact( #"LCS Stop" )
      R_Coil( #Actuator.LCS_OnOff )
   END_RUNG
   // the same network as SCL:
   IF #alwaysON AND #"LCS Start" THEN #Actuator.LCS_OnOff := TRUE; END_IF;
   IF #alwaysON AND #"LCS Stop" THEN #Actuator.LCS_OnOff := FALSE; END_IF;
END_REGION

REGION Network 8: Inload Enable
   RUNG wire#powerrail
      Contact( #alwaysON )
      I_Contact( #State.Tank_HL )
      I_Contact( #"Inload Busy" )
      I_Contact( #State.Tank_inCIP )
      I_Contact( #State.Line_inCIP )
      Coil( #State.Inload_Enable )
   END_RUNG
   // the same network as SCL:
   #State.Inload_Enable := #alwaysON AND NOT #State.Tank_HL AND NOT #"Inload Busy" AND NOT #State.Tank_inCIP AND NOT #State.Line_inCIP;
END_REGION

REGION Network 9: Command Inload Tomato
   RUNG wire#powerrail
      Contact( #alwaysON )
      wire#w1
      Contact( #State.Inload_Enable )
      wire#w2
      Contact( #Cmd.Inload_Tomato )
      wire#w3
      S_Coil( #State.Inloading_Tomato )
   END_RUNG
   RUNG wire#w2
      Contact( #Actuator.LCS_OnOff )
   END_RUNG wire#w3
   RUNG wire#w1
      I_Contact( #State.Inload_Enable )
      R_Coil( #Cmd.Inload_Tomato )
   END_RUNG
   RUNG wire#w1
      I_Contact( #Cmd.Inload_Tomato )
      I_Contact( #Actuator.LCS_OnOff )
      R_Coil( #State.Inloading_Tomato )
   END_RUNG
   // the same network as SCL:
   IF #alwaysON AND #State.Inload_Enable AND (#Cmd.Inload_Tomato OR #Actuator.LCS_OnOff) THEN
       #State.Inloading_Tomato := TRUE;
   END_IF;
   IF #alwaysON AND NOT #State.Inload_Enable THEN #Cmd.Inload_Tomato := FALSE; END_IF;
   IF #alwaysON AND NOT #Cmd.Inload_Tomato AND NOT #Actuator.LCS_OnOff THEN
       #State.Inloading_Tomato := FALSE;
   END_IF;
END_REGION

REGION Network 10: Command Inload Process Water
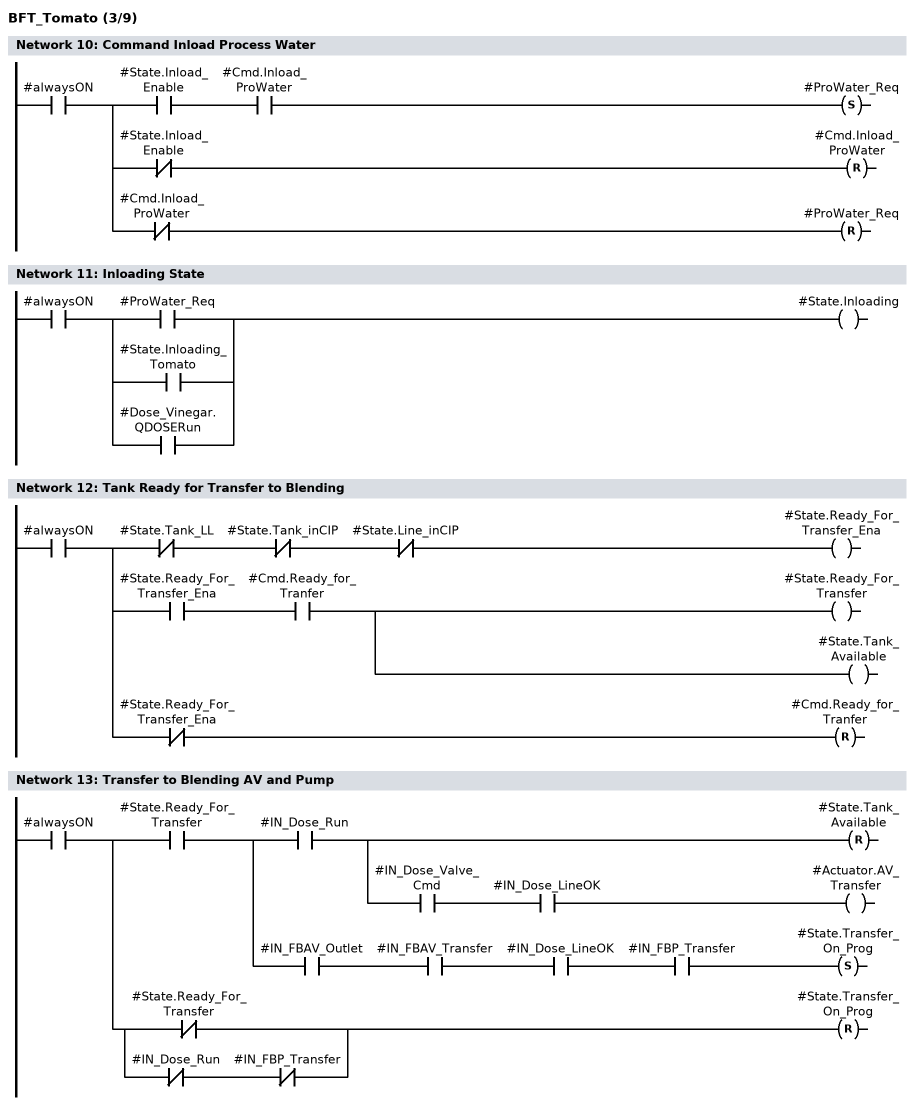
   RUNG wire#powerrail
      Contact( #alwaysON )
      wire#w1
      Contact( #State.Inload_Enable )
      Contact( #Cmd.Inload_ProWater )
      S_Coil( #ProWater_Req )
   END_RUNG
   RUNG wire#w1
      I_Contact( #State.Inload_Enable )
      R_Coil( #Cmd.Inload_ProWater )
   END_RUNG
   RUNG wire#w1
      I_Contact( #Cmd.Inload_ProWater )
      R_Coil( #ProWater_Req )
   END_RUNG
   // the same network as SCL:
   IF #alwaysON AND #State.Inload_Enable AND #Cmd.Inload_ProWater THEN #ProWater_Req := TRUE; END_IF;
   IF #alwaysON AND NOT #State.Inload_Enable THEN #Cmd.Inload_ProWater := FALSE; END_IF;
   IF #alwaysON AND NOT #Cmd.Inload_ProWater THEN #ProWater_Req := FALSE; END_IF;
END_REGION

REGION Network 11: Inloading State
   RUNG wire#powerrail
      Contact( #alwaysON )
      wire#w1
      Contact( #ProWater_Req )
      wire#w2
      Coil( #State.Inloading )
   END_RUNG
   RUNG wire#w1
      Contact( #State.Inloading_Tomato )
   END_RUNG wire#w2
   RUNG wire#w1
      Contact( #Dose_Vinegar.QDOSERun )
   END_RUNG wire#w2
   // the same network as SCL:
   #State.Inloading := #alwaysON AND (#ProWater_Req OR #State.Inloading_Tomato OR #Dose_Vinegar.QDOSERun);
END_REGION

REGION Network 12: Tank Ready for Transfer to Blending
   RUNG wire#powerrail
      Contact( #alwaysON )
      wire#w1
      I_Contact( #State.Tank_LL )
      I_Contact( #State.Tank_inCIP )
      I_Contact( #State.Line_inCIP )
      Coil( #State.Ready_For_Transfer_Ena )
   END_RUNG
   RUNG wire#w1
      Contact( #State.Ready_For_Transfer_Ena )
      Contact( #Cmd.Ready_for_Tranfer )
      wire#w2
      Coil( #State.Ready_For_Transfer )
   END_RUNG
   RUNG wire#w2
      Coil( #State.Tank_Available )
   END_RUNG
   RUNG wire#w1
      I_Contact( #State.Ready_For_Transfer_Ena )
      R_Coil( #Cmd.Ready_for_Tranfer )
   END_RUNG
   // the same network as SCL:
   #State.Ready_For_Transfer_Ena := #alwaysON AND NOT #State.Tank_LL AND NOT #State.Tank_inCIP AND NOT #State.Line_inCIP;
   #State.Ready_For_Transfer := #alwaysON AND #State.Ready_For_Transfer_Ena AND #Cmd.Ready_for_Tranfer;
   #State.Tank_Available := #State.Ready_For_Transfer;
   IF #alwaysON AND NOT #State.Ready_For_Transfer_Ena THEN #Cmd.Ready_for_Tranfer := FALSE; END_IF;
END_REGION

REGION Network 13: Transfer to Blending AV and Pump
   RUNG wire#powerrail
      Contact( #alwaysON )
      wire#w1
      Contact( #State.Ready_For_Transfer )
      wire#w2
      Contact( #IN_Dose_Run )
      wire#w3
      R_Coil( #State.Tank_Available )
   END_RUNG
   RUNG wire#w3
      Contact( #IN_Dose_Valve_Cmd )
      Contact( #IN_Dose_LineOK )
      Coil( #Actuator.AV_Transfer )
   END_RUNG
   RUNG wire#w2
      Contact( #IN_FBAV_Outlet )
      Contact( #IN_FBAV_Transfer )
      Contact( #IN_Dose_LineOK )
      Contact( #IN_FBP_Transfer )
      S_Coil( #State.Transfer_On_Prog )
   END_RUNG
   RUNG wire#w1
      I_Contact( #State.Ready_For_Transfer )
      wire#w4
      R_Coil( #State.Transfer_On_Prog )
   END_RUNG
   RUNG wire#w1
      I_Contact( #IN_Dose_Run )
      I_Contact( #IN_FBP_Transfer )
   END_RUNG wire#w4
   // the same network as SCL:
   #_w1 := #alwaysON AND #State.Ready_For_Transfer;
   #_w2 := #_w1 AND #IN_Dose_Run;
   IF #_w2 THEN #State.Tank_Available := FALSE; END_IF;
   #Actuator.AV_Transfer := #_w2 AND #IN_Dose_Valve_Cmd AND #IN_Dose_LineOK;
   IF #_w1 AND #IN_FBAV_Outlet AND #IN_FBAV_Transfer AND #IN_Dose_LineOK AND #IN_FBP_Transfer THEN
       #State.Transfer_On_Prog := TRUE;
   END_IF;
   IF #alwaysON AND (NOT #State.Ready_For_Transfer OR (NOT #IN_Dose_Run AND NOT #IN_FBP_Transfer)) THEN
       #State.Transfer_On_Prog := FALSE;
   END_IF;
END_REGION

REGION Network 14: Command CIP
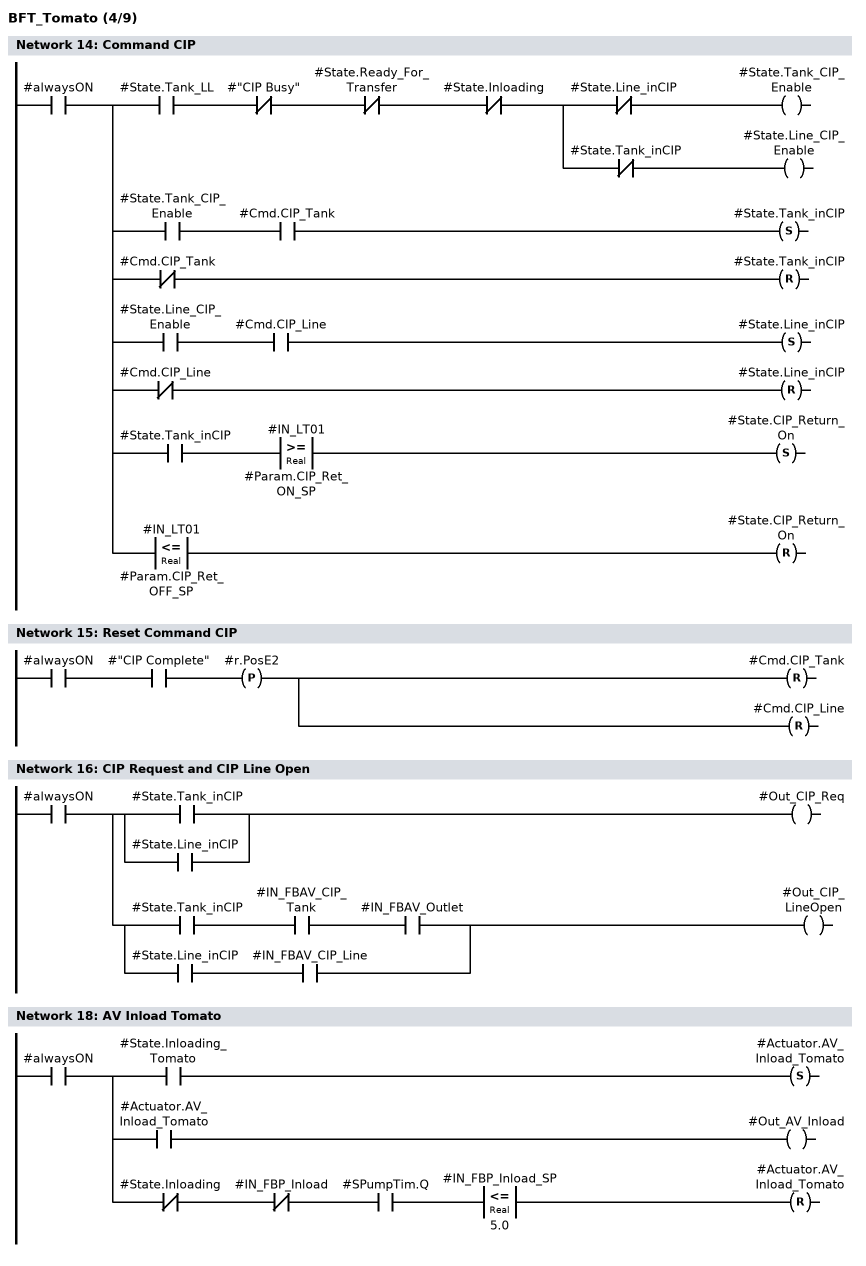
   RUNG wire#powerrail
      Contact( #alwaysON )
      wire#w1
      Contact( #State.Tank_LL )
      I_Contact( #"CIP Busy" )
      I_Contact( #State.Ready_For_Transfer )
      I_Contact( #State.Inloading )
      wire#w2
      I_Contact( #State.Line_inCIP )
      Coil( #State.Tank_CIP_Enable )
   END_RUNG
   RUNG wire#w2
      I_Contact( #State.Tank_inCIP )
      Coil( #State.Line_CIP_Enable )
   END_RUNG
   RUNG wire#w1
      Contact( #State.Tank_CIP_Enable )
      Contact( #Cmd.CIP_Tank )
      S_Coil( #State.Tank_inCIP )
   END_RUNG
   RUNG wire#w1
      I_Contact( #Cmd.CIP_Tank )
      R_Coil( #State.Tank_inCIP )
   END_RUNG
   RUNG wire#w1
      Contact( #State.Line_CIP_Enable )
      Contact( #Cmd.CIP_Line )
      S_Coil( #State.Line_inCIP )
   END_RUNG
   RUNG wire#w1
      I_Contact( #Cmd.CIP_Line )
      R_Coil( #State.Line_inCIP )
   END_RUNG
   RUNG wire#w1
      Contact( #State.Tank_inCIP )
      { S7_Templates := "SrcType := Real" } GE_Contact(in1 := #IN_LT01, in2 := #Param.CIP_Ret_ON_SP)
      S_Coil( #State.CIP_Return_On )
   END_RUNG
   RUNG wire#w1
      { S7_Templates := "SrcType := Real" } LE_Contact(in1 := #IN_LT01, in2 := #Param.CIP_Ret_OFF_SP)
      R_Coil( #State.CIP_Return_On )
   END_RUNG
   // the same network as SCL:
   #_w1 := #alwaysON AND #State.Tank_LL AND NOT #"CIP Busy" AND NOT #State.Ready_For_Transfer AND NOT #State.Inloading;
   #State.Tank_CIP_Enable := #_w1 AND NOT #State.Line_inCIP;
   #State.Line_CIP_Enable := #_w1 AND NOT #State.Tank_inCIP;
   IF #alwaysON AND #State.Tank_CIP_Enable AND #Cmd.CIP_Tank THEN #State.Tank_inCIP := TRUE; END_IF;
   IF #alwaysON AND NOT #Cmd.CIP_Tank THEN #State.Tank_inCIP := FALSE; END_IF;
   IF #alwaysON AND #State.Line_CIP_Enable AND #Cmd.CIP_Line THEN #State.Line_inCIP := TRUE; END_IF;
   IF #alwaysON AND NOT #Cmd.CIP_Line THEN #State.Line_inCIP := FALSE; END_IF;
   IF #alwaysON AND #State.Tank_inCIP AND (#IN_LT01 >= #Param.CIP_Ret_ON_SP) THEN
       #State.CIP_Return_On := TRUE;
   END_IF;
   IF #alwaysON AND (#IN_LT01 <= #Param.CIP_Ret_OFF_SP) THEN #State.CIP_Return_On := FALSE; END_IF;
END_REGION

REGION Network 15: Reset Command CIP
   RUNG wire#powerrail
      Contact( #alwaysON )
      Contact( #"CIP Complete" )
      P_Trig( #r.PosE2 )
      wire#w1
      R_Coil( #Cmd.CIP_Tank )
   END_RUNG
   RUNG wire#w1
      R_Coil( #Cmd.CIP_Line )
   END_RUNG
   // the same network as SCL:
   #_w1 := #alwaysON AND #"CIP Complete";
   #_w2 := #_w1 AND NOT #r.PosE2;   // rising edge
   #r.PosE2 := #_w1;
   IF #_w2 THEN
       #Cmd.CIP_Tank := FALSE;
       #Cmd.CIP_Line := FALSE;
   END_IF;
END_REGION

REGION Network 16: CIP Request and CIP Line Open
   RUNG wire#powerrail
      Contact( #alwaysON )
      wire#w1
      Contact( #State.Tank_inCIP )
      wire#w2
      Coil( #Out_CIP_Req )
   END_RUNG
   RUNG wire#w1
      Contact( #State.Line_inCIP )
   END_RUNG wire#w2
   RUNG wire#w1
      Contact( #State.Tank_inCIP )
      Contact( #IN_FBAV_CIP_Tank )
      Contact( #IN_FBAV_Outlet )
      wire#w3
      Coil( #Out_CIP_LineOpen )
   END_RUNG
   RUNG wire#w1
      Contact( #State.Line_inCIP )
      Contact( #IN_FBAV_CIP_Line )
   END_RUNG wire#w3
   // the same network as SCL:
   #Out_CIP_Req := #alwaysON AND (#State.Tank_inCIP OR #State.Line_inCIP);
   #Out_CIP_LineOpen := #alwaysON AND ((#State.Tank_inCIP AND #IN_FBAV_CIP_Tank AND #IN_FBAV_Outlet) OR (#State.Line_inCIP AND #IN_FBAV_CIP_Line));
END_REGION

REGION Network 18: AV Inload Tomato
   RUNG wire#powerrail
      Contact( #alwaysON )
      wire#w1
      Contact( #State.Inloading_Tomato )
      S_Coil( #Actuator.AV_Inload_Tomato )
   END_RUNG
   RUNG wire#w1
      Contact( #Actuator.AV_Inload_Tomato )
      Coil( #Out_AV_Inload )
   END_RUNG
   RUNG wire#w1
      I_Contact( #State.Inloading )
      I_Contact( #IN_FBP_Inload )
      Contact( #SPumpTim.Q )
      { S7_Templates := "SrcType := Real" } LE_Contact(in1 := #IN_FBP_Inload_SP, in2 := 5.0)
      R_Coil( #Actuator.AV_Inload_Tomato )
   END_RUNG
   // the same network as SCL:
   IF #alwaysON AND #State.Inloading_Tomato THEN #Actuator.AV_Inload_Tomato := TRUE; END_IF;
   #Out_AV_Inload := #alwaysON AND #Actuator.AV_Inload_Tomato;
   IF #alwaysON AND NOT #State.Inloading AND NOT #IN_FBP_Inload AND #SPumpTim.Q AND (#IN_FBP_Inload_SP <= 5.0) THEN
       #Actuator.AV_Inload_Tomato := FALSE;
   END_IF;
END_REGION

REGION Network 19: AV Inload ProWater
